LIN {X 0,Y 538.13,Z 595.444,A -85,B 0,C 180,E1 -4149.775,E2 -4149.775} C_VEL
LIN {X 0,Y 538.366,Z 585.113,A -85,B 0,C 180,E1 -4150.721,E2 -4150.721} C_VEL
LIN {X 0,Y 538.641,Z 573.919,A -85,B 0,C 180,E1 -4151.54,E2 -4151.54} C_VEL
LIN {X 0,Y 538.832,Z 561.69,A -85,B 0,C 180,E1 -4152.237,E2 -4152.237} C_VEL
LIN {X 0,Y 539.079,Z 549.655,A -85,B 0,C 180,E1 -4152.757,E2 -4152.757} C_VEL
LIN {X 0,Y 539.25,Z 536.276,A -85,B 0,C 180,E1 -4153.16,E2 -4153.16} C_VEL
LIN {X 0,Y 539.341,Z 523.449,A -85,B 0,C 180,E1 -4153.397,E2 -4153.397} C_VEL
LIN {X 0,Y 539.592,Z 428.794,A -85,B 0,C 180,E1 -4154.665,E2 -4154.665} C_VEL
LIN {X 0,Y 538.556,Z 421.341,A -85,B 0,C 180,E1 -4154.818,E2 -4154.818} C_VEL
LIN {X 0,Y 538.888,Z 398.914,A -85,B 0,C 180,E1 -4157.681,E2 -4157.681} C_VEL
LIN {X 0,Y 539.305,Z 376.337,A -85,B 0,C 180,E1 -4160.601,E2 -4160.601} C_VEL
LIN {X 0,Y 539.597,Z 359.195,A -85,B 0,C 180,E1 -4162.827,E2 -4162.827} C_VEL
LIN {X 0,Y 539.121,Z 355.573,A -85,B 0,C 180,E1 -4163.32,E2 -4163.32} C_VEL
LIN {X 0,Y 536.659,Z 349.989,A -85,B 0,C 180,E1 -4164.149,E2 -4164.149} C_VEL
LIN {X 0,Y 533.324,Z 343.375,A -85,B 0,C 180,E1 -4165.16,E2 -4165.16} C_VEL
LIN {X 0,Y 532.661,Z 341.028,A -85,B 0,C 180,E1 -4165.499,E2 -4165.499} C_VEL
LIN {X 0,Y 531.046,Z 333.084,A -85,B 0,C 180,E1 -4166.66,E2 -4166.66} C_VEL
LIN {X 0,Y 530.987,Z 332.967,A -85,B 0,C 180,E1 -4169.322,E2 -4169.322} C_VEL
LIN {X 0,Y 530.971,Z 332.971,A -85,B 0,C 180,E1 -4172.1,E2 -4172.1} C_VEL
LIN {X 0,Y 530.975,Z 332.968,A -85,B 0,C 180,E1 -4174.851,E2 -4174.851} C_VEL
LIN {X 0,Y 530.97,Z 332.966,A -85,B 0,C 180,E1 -4177.507,E2 -4177.507} C_VEL
LIN {X 0,Y 530.986,Z 332.97,A -85,B 0,C 180,E1 -4180.433,E2 -4180.433} C_VEL
LIN {X 0,Y 530.966,Z 332.964,A -85,B 0,C 180,E1 -4183.281,E2 -4183.281} C_VEL
LIN {X 0,Y 530.986,Z 332.959,A -85,B 0,C 180,E1 -4185.621,E2 -4185.621} C_VEL
LIN {X 0,Y 530.998,Z 332.964,A -85,B 0,C 180,E1 -4188.564,E2 -4188.564} C_VEL
LIN {X 0,Y 530.962,Z 332.967,A -85,B 0,C 180,E1 -4191.529,E2 -4191.529} C_VEL
LIN {X 0,Y 530.982,Z 332.968,A -85,B 0,C 180,E1 -4194.381,E2 -4194.381} C_VEL
LIN {X 0,Y 530.972,Z 332.964,A -85,B 0,C 180,E1 -4197.133,E2 -4197.133} C_VEL
LIN {X 0,Y 530.975,Z 332.967,A -85,B 0,C 180,E1 -4199.803,E2 -4199.803} C_VEL
LIN {X 0,Y 531.021,Z 332.964,A -85,B 0,C 180,E1 -4202.466,E2 -4202.466} C_VEL
LIN {X 0,Y 531.02,Z 332.968,A -85,B 0,C 180,E1 -4205.569,E2 -4205.569} C_VEL
LIN {X 0,Y 531.055,Z 333.297,A -85,B 0,C 180,E1 -4205.844,E2 -4205.844} C_VEL
LIN {X 0,Y 532.646,Z 342.082,A -85,B 0,C 180,E1 -4207.318,E2 -4207.318} C_VEL
LIN {X 0,Y 532.073,Z 361.559,A -85,B 0,C 180,E1 -4210.316,E2 -4210.316} C_VEL
LIN {X 0,Y 531.85,Z 372.04,A -85,B 0,C 180,E1 -4211.889,E2 -4211.889} C_VEL
LIN {X 0,Y 532.504,Z 375.809,A -85,B 0,C 180,E1 -4212.004,E2 -4212.004} C_VEL
LIN {X 0,Y 533.949,Z 384.074,A -85,B 0,C 180,E1 -4212.169,E2 -4212.169} C_VEL
LIN {X 0,Y 533.298,Z 508.609,A -85,B 0,C 180,E1 -4213.884,E2 -4213.884} C_VEL
LIN {X 0,Y 533.064,Z 523.105,A -85,B 0,C 180,E1 -4214.225,E2 -4214.225} C_VEL
LIN {X 0,Y 532.771,Z 537.785,A -85,B 0,C 180,E1 -4214.751,E2 -4214.751} C_VEL
LIN {X 0,Y 532.511,Z 550.755,A -85,B 0,C 180,E1 -4215.379,E2 -4215.379} C_VEL
LIN {X 0,Y 532.156,Z 561.953,A -85,B 0,C 180,E1 -4216.052,E2 -4216.052} C_VEL
LIN {X 0,Y 531.811,Z 573.767,A -85,B 0,C 180,E1 -4216.919,E2 -4216.919} C_VEL
LIN {X 0,Y 531.434,Z 586.265,A -85,B 0,C 180,E1 -4218.057,E2 -4218.057} C_VEL
LIN {X 0,Y 531.191,Z 595.879,A -85,B 0,C 180,E1 -4219.132,E2 -4219.132} C_VEL
LIN {X 0,Y 530.938,Z 603.182,A -85,B 0,C 180,E1 -4220.09,E2 -4220.09} C_VEL
LIN {X 0,Y 530.824,Z 609.461,A -85,B 0,C 180,E1 -4221.049,E2 -4221.049} C_VEL
LIN {X 0,Y 530.706,Z 614.868,A -85,B 0,C 180,E1 -4222.006,E2 -4222.006} C_VEL
LIN {X 0,Y 530.575,Z 620.295,A -85,B 0,C 180,E1 -4223.152,E2 -4223.152} C_VEL
LIN {X 0,Y 530.567,Z 624.738,A -85,B 0,C 180,E1 -4224.298,E2 -4224.298} C_VEL
LIN {X 0,Y 530.449,Z 628.286,A -85,B 0,C 180,E1 -4225.44,E2 -4225.44} C_VEL
LIN {X 0,Y 530.497,Z 630.208,A -85,B 0,C 180,E1 -4226.201,E2 -4226.201} C_VEL
LIN {X 0,Y 530.41,Z 632.929,A -85,B 0,C 180,E1 -4227.721,E2 -4227.721} C_VEL
LIN {X 0,Y 530.34,Z 634.237,A -85,B 0,C 180,E1 -4229.24,E2 -4229.24} C_VEL
LIN {X 0,Y 530.342,Z 634.496,A -85,B 0,C 180,E1 -4229.999,E2 -4229.999} C_VEL
LIN {X 0,Y 530.357,Z 633.834,A -85,B 0,C 180,E1 -4231.518,E2 -4231.518} C_VEL
LIN {X 0,Y 530.451,Z 631.843,A -85,B 0,C 180,E1 -4233.037,E2 -4233.037} C_VEL
LIN {X 0,Y 530.497,Z 630.435,A -85,B 0,C 180,E1 -4233.797,E2 -4233.797} C_VEL
LIN {X 0,Y 530.514,Z 626.296,A -85,B 0,C 180,E1 -4235.32,E2 -4235.32} C_VEL
LIN {X 0,Y 530.555,Z 623.773,A -85,B 0,C 180,E1 -4236.082,E2 -4236.082} C_VEL
LIN {X 0,Y 530.584,Z 619.088,A -85,B 0,C 180,E1 -4237.228,E2 -4237.228} C_VEL
LIN {X 0,Y 530.774,Z 612.262,A -85,B 0,C 180,E1 -4238.566,E2 -4238.566} C_VEL
LIN {X 0,Y 530.895,Z 605.147,A -85,B 0,C 180,E1 -4239.716,E2 -4239.716} C_VEL
LIN {X 0,Y 531.097,Z 598.173,A -85,B 0,C 180,E1 -4240.675,E2 -4240.675} C_VEL
LIN {X 0,Y 531.373,Z 589.079,A -85,B 0,C 180,E1 -4241.733,E2 -4241.733} C_VEL
LIN {X 0,Y 531.625,Z 580.332,A -85,B 0,C 180,E1 -4242.598,E2 -4242.598} C_VEL
LIN {X 0,Y 531.914,Z 569.995,A -85,B 0,C 180,E1 -4243.465,E2 -4243.465} C_VEL
LIN {X 0,Y 532.249,Z 558.953,A -85,B 0,C 180,E1 -4244.236,E2 -4244.236} C_VEL
LIN {X 0,Y 532.596,Z 544.118,A -85,B 0,C 180,E1 -4245.057,E2 -4245.057} C_VEL
LIN {X 0,Y 532.936,Z 531.187,A -85,B 0,C 180,E1 -4245.595,E2 -4245.595} C_VEL
LIN {X 0,Y 533.153,Z 518.305,A -85,B 0,C 180,E1 -4245.992,E2 -4245.992} C_VEL
LIN {X 0,Y 533.333,Z 505.438,A -85,B 0,C 180,E1 -4246.26,E2 -4246.26} C_VEL
LIN {X 0,Y 533.841,Z 382.931,A -85,B 0,C 180,E1 -4247.941,E2 -4247.941} C_VEL
LIN {X 0,Y 531.872,Z 372.407,A -85,B 0,C 180,E1 -4248.173,E2 -4248.173} C_VEL
LIN {X 0,Y 531.921,Z 368.698,A -85,B 0,C 180,E1 -4248.686,E2 -4248.686} C_VEL
LIN {X 0,Y 532.441,Z 349.078,A -85,B 0,C 180,E1 -4251.689,E2 -4251.689} C_VEL
LIN {X 0,Y 532.622,Z 341.232,A -85,B 0,C 180,E1 -4252.906,E2 -4252.906} C_VEL
LIN {X 0,Y 531.016,Z 333.185,A -85,B 0,C 180,E1 -4254.273,E2 -4254.273} C_VEL
LIN {X 0,Y 531.014,Z 332.957,A -85,B 0,C 180,E1 -4255.896,E2 -4255.896} C_VEL
LIN {X 0,Y 530.998,Z 332.957,A -85,B 0,C 180,E1 -4258.454,E2 -4258.454} C_VEL
LIN {X 0,Y 530.965,Z 332.967,A -85,B 0,C 180,E1 -4261.077,E2 -4261.077} C_VEL
LIN {X 0,Y 530.99,Z 332.966,A -85,B 0,C 180,E1 -4263.771,E2 -4263.771} C_VEL
LIN {X 0,Y 530.965,Z 332.968,A -85,B 0,C 180,E1 -4266.556,E2 -4266.556} C_VEL
LIN {X 0,Y 531.002,Z 332.964,A -85,B 0,C 180,E1 -4269.856,E2 -4269.856} C_VEL
LIN {X 0,Y 530.977,Z 332.967,A -85,B 0,C 180,E1 -4272.455,E2 -4272.455} C_VEL
LIN {X 0,Y 530.982,Z 332.962,A -85,B 0,C 180,E1 -4275.62,E2 -4275.62} C_VEL
LIN {X 0,Y 531.013,Z 332.961,A -85,B 0,C 180,E1 -4278.566,E2 -4278.566} C_VEL
LIN {X 0,Y 530.953,Z 332.967,A -85,B 0,C 180,E1 -4281.529,E2 -4281.529} C_VEL
LIN {X 0,Y 530.974,Z 332.964,A -85,B 0,C 180,E1 -4284.381,E2 -4284.381} C_VEL
LIN {X 0,Y 530.967,Z 332.968,A -85,B 0,C 180,E1 -4287.133,E2 -4287.133} C_VEL
LIN {X 0,Y 530.977,Z 332.958,A -85,B 0,C 180,E1 -4289.803,E2 -4289.803} C_VEL
LIN {X 0,Y 531.009,Z 332.953,A -85,B 0,C 180,E1 -4292.465,E2 -4292.465} C_VEL
LIN {X 0,Y 531.001,Z 332.962,A -85,B 0,C 180,E1 -4294.942,E2 -4294.942} C_VEL
LIN {X 0,Y 530.982,Z 332.963,A -85,B 0,C 180,E1 -4297.893,E2 -4297.893} C_VEL
LIN {X 0,Y 530.988,Z 332.963,A -85,B 0,C 180,E1 -4300.677,E2 -4300.677} C_VEL
LIN {X 0,Y 530.985,Z 332.968,A -85,B 0,C 180,E1 -4303.071,E2 -4303.071} C_VEL
LIN {X 0,Y 531.03,Z 332.963,A -85,B 0,C 180,E1 -4305.436,E2 -4305.436} C_VEL
LIN {X 0,Y 531.043,Z 332.956,A -85,B 0,C 180,E1 -4308.55,E2 -4308.55} C_VEL
LIN {X 0,Y 531.052,Z 332.956,A -85,B 0,C 180,E1 -4311.629,E2 -4311.629} C_VEL
LIN {X 0,Y 531.132,Z 332.947,A -85,B 0,C 180,E1 -4314.685,E2 -4314.685} C_VEL
LIN {X 0,Y 531.131,Z 332.944,A -85,B 0,C 180,E1 -4317.725,E2 -4317.725} C_VEL
LIN {X 0,Y 531.149,Z 332.948,A -85,B 0,C 180,E1 -4320.758,E2 -4320.758} C_VEL
LIN {X 0,Y 531.103,Z 332.952,A -85,B 0,C 180,E1 -4323.034,E2 -4323.034} C_VEL
LIN {X 0,Y 531.076,Z 332.952,A -85,B 0,C 180,E1 -4326.077,E2 -4326.077} C_VEL
LIN {X 0,Y 531.028,Z 332.957,A -85,B 0,C 180,E1 -4329.138,E2 -4329.138} C_VEL
LIN {X 0,Y 531.051,Z 332.954,A -85,B 0,C 180,E1 -4331.678,E2 -4331.678} C_VEL
LIN {X 0,Y 531.019,Z 332.959,A -85,B 0,C 180,E1 -4334.956,E2 -4334.956} C_VEL
LIN {X 0,Y 531.006,Z 332.96,A -85,B 0,C 180,E1 -4337.723,E2 -4337.723} C_VEL
LIN {X 0,Y 530.995,Z 332.963,A -85,B 0,C 180,E1 -4340.938,E2 -4340.938} C_VEL
LIN {X 0,Y 530.998,Z 332.964,A -85,B 0,C 180,E1 -4344.046,E2 -4344.046} C_VEL
LIN {X 0,Y 531.002,Z 332.959,A -85,B 0,C 180,E1 -4346.744,E2 -4346.744} C_VEL
LIN {X 0,Y 530.973,Z 332.952,A -85,B 0,C 180,E1 -4349.323,E2 -4349.323} C_VEL
LIN {X 0,Y 530.972,Z 332.966,A -85,B 0,C 180,E1 -4352.104,E2 -4352.104} C_VEL
LIN {X 0,Y 530.982,Z 332.965,A -85,B 0,C 180,E1 -4354.855,E2 -4354.855} C_VEL
LIN {X 0,Y 530.958,Z 332.958,A -85,B 0,C 180,E1 -4357.508,E2 -4357.508} C_VEL
LIN {X 0,Y 531.02,Z 332.966,A -85,B 0,C 180,E1 -4360.429,E2 -4360.429} C_VEL
LIN {X 0,Y 530.961,Z 332.965,A -85,B 0,C 180,E1 -4363.495,E2 -4363.495} C_VEL
LIN {X 0,Y 530.959,Z 332.971,A -85,B 0,C 180,E1 -4366.507,E2 -4366.507} C_VEL
LIN {X 0,Y 531.021,Z 332.96,A -85,B 0,C 180,E1 -4369.572,E2 -4369.572} C_VEL
LIN {X 0,Y 530.964,Z 332.968,A -85,B 0,C 180,E1 -4372.578,E2 -4372.578} C_VEL
LIN {X 0,Y 531.001,Z 332.963,A -85,B 0,C 180,E1 -4375.313,E2 -4375.313} C_VEL
LIN {X 0,Y 530.98,Z 332.972,A -85,B 0,C 180,E1 -4378.034,E2 -4378.034} C_VEL
LIN {X 0,Y 531.004,Z 332.951,A -85,B 0,C 180,E1 -4380.872,E2 -4380.872} C_VEL
LIN {X 0,Y 531.01,Z 332.966,A -85,B 0,C 180,E1 -4383.258,E2 -4383.258} C_VEL
LIN {X 0,Y 531.009,Z 333.054,A -85,B 0,C 180,E1 -4385.726,E2 -4385.726} C_VEL
LIN {X 0,Y 532.599,Z 340.946,A -85,B 0,C 180,E1 -4387.092,E2 -4387.092} C_VEL
LIN {X 0,Y 532.226,Z 357.451,A -85,B 0,C 180,E1 -4389.644,E2 -4389.644} C_VEL
LIN {X 0,Y 531.845,Z 372.091,A -85,B 0,C 180,E1 -4391.849,E2 -4391.849} C_VEL
LIN {X 0,Y 532.716,Z 376.892,A -85,B 0,C 180,E1 -4391.982,E2 -4391.982} C_VEL
LIN {X 0,Y 533.891,Z 384.047,A -85,B 0,C 180,E1 -4392.122,E2 -4392.122} C_VEL
LIN {X 0,Y 533.278,Z 508.696,A -85,B 0,C 180,E1 -4393.836,E2 -4393.836} C_VEL
LIN {X 0,Y 533.082,Z 523.313,A -85,B 0,C 180,E1 -4394.188,E2 -4394.188} C_VEL
LIN {X 0,Y 532.852,Z 536.169,A -85,B 0,C 180,E1 -4394.639,E2 -4394.639} C_VEL
LIN {X 0,Y 532.521,Z 549.89,A -85,B 0,C 180,E1 -4395.284,E2 -4395.284} C_VEL
LIN {X 0,Y 532.144,Z 562.69,A -85,B 0,C 180,E1 -4396.054,E2 -4396.054} C_VEL
LIN {X 0,Y 531.803,Z 574.318,A -85,B 0,C 180,E1 -4396.921,E2 -4396.921} C_VEL
LIN {X 0,Y 531.453,Z 585.317,A -85,B 0,C 180,E1 -4397.917,E2 -4397.917} C_VEL
LIN {X 0,Y 531.234,Z 594.715,A -85,B 0,C 180,E1 -4398.942,E2 -4398.942} C_VEL
LIN {X 0,Y 530.935,Z 603.563,A -85,B 0,C 180,E1 -4400.092,E2 -4400.092} C_VEL
LIN {X 0,Y 530.774,Z 612.04,A -85,B 0,C 180,E1 -4401.434,E2 -4401.434} C_VEL
LIN {X 0,Y 530.585,Z 618.866,A -85,B 0,C 180,E1 -4402.772,E2 -4402.772} C_VEL
LIN {X 0,Y 530.584,Z 624.962,A -85,B 0,C 180,E1 -4404.3,E2 -4404.3} C_VEL
LIN {X 0,Y 530.449,Z 628.449,A -85,B 0,C 180,E1 -4405.441,E2 -4405.441} C_VEL
LIN {X 0,Y 530.452,Z 631.838,A -85,B 0,C 180,E1 -4406.963,E2 -4406.963} C_VEL
LIN {X 0,Y 530.357,Z 633.838,A -85,B 0,C 180,E1 -4408.482,E2 -4408.482} C_VEL
LIN {X 0,Y 530.341,Z 634.5,A -85,B 0,C 180,E1 -4410.001,E2 -4410.001} C_VEL
LIN {X 0,Y 530.357,Z 633.834,A -85,B 0,C 180,E1 -4411.52,E2 -4411.52} C_VEL
LIN {X 0,Y 530.452,Z 631.83,A -85,B 0,C 180,E1 -4413.039,E2 -4413.039} C_VEL
LIN {X 0,Y 530.449,Z 628.441,A -85,B 0,C 180,E1 -4414.56,E2 -4414.56} C_VEL
LIN {X 0,Y 530.561,Z 623.565,A -85,B 0,C 180,E1 -4416.084,E2 -4416.084} C_VEL
LIN {X 0,Y 530.642,Z 617.05,A -85,B 0,C 180,E1 -4417.612,E2 -4417.612} C_VEL
LIN {X 0,Y 530.812,Z 609.797,A -85,B 0,C 180,E1 -4418.951,E2 -4418.951} C_VEL
LIN {X 0,Y 531.018,Z 600.815,A -85,B 0,C 180,E1 -4420.293,E2 -4420.293} C_VEL
LIN {X 0,Y 531.312,Z 591.383,A -85,B 0,C 180,E1 -4421.445,E2 -4421.445} C_VEL
LIN {X 0,Y 531.586,Z 580.942,A -85,B 0,C 180,E1 -4422.504,E2 -4422.504} C_VEL
LIN {X 0,Y 531.951,Z 569.413,A -85,B 0,C 180,E1 -4423.466,E2 -4423.466} C_VEL
LIN {X 0,Y 532.284,Z 558.201,A -85,B 0,C 180,E1 -4424.237,E2 -4424.237} C_VEL
LIN {X 0,Y 532.613,Z 546.119,A -85,B 0,C 180,E1 -4424.911,E2 -4424.911} C_VEL
LIN {X 0,Y 532.939,Z 533.26,A -85,B 0,C 180,E1 -4425.473,E2 -4425.473} C_VEL
LIN {X 0,Y 533.092,Z 519.619,A -85,B 0,C 180,E1 -4425.916,E2 -4425.916} C_VEL
LIN {X 0,Y 533.304,Z 505.572,A -85,B 0,C 180,E1 -4426.214,E2 -4426.214} C_VEL
LIN {X 0,Y 533.922,Z 383.42,A -85,B 0,C 180,E1 -4427.886,E2 -4427.886} C_VEL
LIN {X 0,Y 531.879,Z 372.396,A -85,B 0,C 180,E1 -4428.129,E2 -4428.129} C_VEL
LIN {X 0,Y 531.938,Z 367.082,A -85,B 0,C 180,E1 -4428.887,E2 -4428.887} C_VEL
LIN {X 0,Y 532.429,Z 348.776,A -85,B 0,C 180,E1 -4431.692,E2 -4431.692} C_VEL
LIN {X 0,Y 532.605,Z 340.932,A -85,B 0,C 180,E1 -4432.909,E2 -4432.909} C_VEL
LIN {X 0,Y 531.04,Z 333.202,A -85,B 0,C 180,E1 -4434.222,E2 -4434.222} C_VEL
LIN {X 0,Y 531.011,Z 332.961,A -85,B 0,C 180,E1 -4435.058,E2 -4435.058} C_VEL
LIN {X 0,Y 531.022,Z 332.964,A -85,B 0,C 180,E1 -4437.596,E2 -4437.596} C_VEL
LIN {X 0,Y 530.979,Z 332.968,A -85,B 0,C 180,E1 -4440.646,E2 -4440.646} C_VEL
LIN {X 0,Y 530.995,Z 332.968,A -85,B 0,C 180,E1 -4443.773,E2 -4443.773} C_VEL
LIN {X 0,Y 530.974,Z 332.968,A -85,B 0,C 180,E1 -4446.558,E2 -4446.558} C_VEL
LIN {X 0,Y 530.983,Z 332.971,A -85,B 0,C 180,E1 -4449.854,E2 -4449.854} C_VEL
LIN {X 0,Y 530.982,Z 332.966,A -85,B 0,C 180,E1 -4452.457,E2 -4452.457} C_VEL
LIN {X 0,Y 530.987,Z 332.969,A -85,B 0,C 180,E1 -4455.622,E2 -4455.622} C_VEL
LIN {X 0,Y 531.001,Z 332.964,A -85,B 0,C 180,E1 -4458.565,E2 -4458.565} C_VEL
LIN {X 0,Y 530.961,Z 332.973,A -85,B 0,C 180,E1 -4461.53,E2 -4461.53} C_VEL
LIN {X 0,Y 530.958,Z 332.969,A -85,B 0,C 180,E1 -4464.38,E2 -4464.38} C_VEL
LIN {X 0,Y 530.972,Z 332.97,A -85,B 0,C 180,E1 -4467.134,E2 -4467.134} C_VEL
LIN {X 0,Y 530.974,Z 332.973,A -85,B 0,C 180,E1 -4469.803,E2 -4469.803} C_VEL
LIN {X 0,Y 531.02,Z 332.964,A -85,B 0,C 180,E1 -4472.467,E2 -4472.467} C_VEL
LIN {X 0,Y 531.038,Z 333.152,A -85,B 0,C 180,E1 -4473.857,E2 -4473.857} C_VEL
LIN {X 0,Y 532.577,Z 341.879,A -85,B 0,C 180,E1 -4475.021,E2 -4475.021} C_VEL
LIN {X 0,Y 532.429,Z 361.787,A -85,B 0,C 180,E1 -4477.518,E2 -4477.518} C_VEL
LIN {X 0,Y 532.201,Z 380.833,A -85,B 0,C 180,E1 -4479.919,E2 -4479.919} C_VEL
LIN {X 0,Y 531.914,Z 397.433,A -85,B 0,C 180,E1 -4482.049,E2 -4482.049} C_VEL
LIN {X 0,Y 531.596,Z 417.775,A -85,B 0,C 180,E1 -4484.668,E2 -4484.668} C_VEL
LIN {X 0,Y 531.551,Z 421.298,A -85,B 0,C 180,E1 -4485.083,E2 -4485.083} C_VEL
LIN {X 0,Y 532.8,Z 431.144,A -85,B 0,C 180,E1 -4485.276,E2 -4485.276} C_VEL
LIN {X 0,Y 532.344,Z 530.888,A -85,B 0,C 180,E1 -4486.666,E2 -4486.666} C_VEL
LIN {X 0,Y 532.209,Z 543.359,A -85,B 0,C 180,E1 -4486.979,E2 -4486.979} C_VEL
LIN {X 0,Y 531.963,Z 556.15,A -85,B 0,C 180,E1 -4487.458,E2 -4487.458} C_VEL
LIN {X 0,Y 531.746,Z 568.289,A -85,B 0,C 180,E1 -4488.076,E2 -4488.076} C_VEL
LIN {X 0,Y 531.523,Z 578.707,A -85,B 0,C 180,E1 -4488.754,E2 -4488.754} C_VEL
LIN {X 0,Y 531.25,Z 589.326,A -85,B 0,C 180,E1 -4489.616,E2 -4489.616} C_VEL
LIN {X 0,Y 531.006,Z 599.735,A -85,B 0,C 180,E1 -4490.669,E2 -4490.669} C_VEL
LIN {X 0,Y 530.857,Z 607.422,A -85,B 0,C 180,E1 -4491.626,E2 -4491.626} C_VEL
LIN {X 0,Y 530.673,Z 614.918,A -85,B 0,C 180,E1 -4492.772,E2 -4492.772} C_VEL
LIN {X 0,Y 530.611,Z 620.932,A -85,B 0,C 180,E1 -4493.918,E2 -4493.918} C_VEL
LIN {X 0,Y 530.459,Z 625.687,A -85,B 0,C 180,E1 -4495.06,E2 -4495.06} C_VEL
LIN {X 0,Y 530.517,Z 629.324,A -85,B 0,C 180,E1 -4496.202,E2 -4496.202} C_VEL
LIN {X 0,Y 530.458,Z 631.196,A -85,B 0,C 180,E1 -4496.962,E2 -4496.962} C_VEL
LIN {X 0,Y 530.411,Z 632.631,A -85,B 0,C 180,E1 -4497.722,E2 -4497.722} C_VEL
LIN {X 0,Y 530.344,Z 634.256,A -85,B 0,C 180,E1 -4499.241,E2 -4499.241} C_VEL
LIN {X 0,Y 530.343,Z 634.497,A -85,B 0,C 180,E1 -4500,E2 -4500} C_VEL
LIN {X 0,Y 530.344,Z 634.312,A -85,B 0,C 180,E1 -4500.759,E2 -4500.759} C_VEL
LIN {X 0,Y 530.41,Z 632.763,A -85,B 0,C 180,E1 -4502.278,E2 -4502.278} C_VEL
LIN {X 0,Y 530.458,Z 631.4,A -85,B 0,C 180,E1 -4503.038,E2 -4503.038} C_VEL
LIN {X 0,Y 530.523,Z 628.526,A -85,B 0,C 180,E1 -4504.178,E2 -4504.178} C_VEL
LIN {X 0,Y 530.524,Z 624.616,A -85,B 0,C 180,E1 -4505.321,E2 -4505.321} C_VEL
LIN {X 0,Y 530.606,Z 618.542,A -85,B 0,C 180,E1 -4506.66,E2 -4506.66} C_VEL
LIN {X 0,Y 530.759,Z 611.965,A -85,B 0,C 180,E1 -4507.801,E2 -4507.801} C_VEL
LIN {X 0,Y 530.907,Z 603.733,A -85,B 0,C 180,E1 -4508.948,E2 -4508.948} C_VEL
LIN {X 0,Y 531.098,Z 595.256,A -85,B 0,C 180,E1 -4509.906,E2 -4509.906} C_VEL
LIN {X 0,Y 531.377,Z 584.867,A -85,B 0,C 180,E1 -4510.864,E2 -4510.864} C_VEL
LIN {X 0,Y 531.636,Z 574.017,A -85,B 0,C 180,E1 -4511.667,E2 -4511.667} C_VEL
LIN {X 0,Y 531.832,Z 563.162,A -85,B 0,C 180,E1 -4512.303,E2 -4512.303} C_VEL
LIN {X 0,Y 532.104,Z 550.353,A -85,B 0,C 180,E1 -4512.879,E2 -4512.879} C_VEL
LIN {X 0,Y 532.292,Z 537.451,A -85,B 0,C 180,E1 -4513.287,E2 -4513.287} C_VEL
LIN {X 0,Y 532.416,Z 523.828,A -85,B 0,C 180,E1 -4513.551,E2 -4513.551} C_VEL
LIN {X 0,Y 532.692,Z 429.041,A -85,B 0,C 180,E1 -4514.851,E2 -4514.851} C_VEL
LIN {X 0,Y 531.559,Z 421.111,A -85,B 0,C 180,E1 -4515.025,E2 -4515.025} C_VEL
LIN {X 0,Y 532.009,Z 396.96,A -85,B 0,C 180,E1 -4518.151,E2 -4518.151} C_VEL
LIN {X 0,Y 532.469,Z 371.438,A -85,B 0,C 180,E1 -4521.486,E2 -4521.486} C_VEL
LIN {X 0,Y 532.901,Z 351.257,A -85,B 0,C 180,E1 -4524.132,E2 -4524.132} C_VEL
LIN {X 0,Y 532.82,Z 341.844,A -85,B 0,C 180,E1 -4525.384,E2 -4525.384} C_VEL
LIN {X 0,Y 532.661,Z 341.028,A -85,B 0,C 180,E1 -4525.499,E2 -4525.499} C_VEL
LIN {X 0,Y 531.517,Z 338.82,A -85,B 0,C 180,E1 -4525.844,E2 -4525.844} C_VEL
LIN {X 0,Y 528.005,Z 335.837,A -85,B 0,C 180,E1 -4526.408,E2 -4526.408} C_VEL
LIN {X 0,Y 524.989,Z 334.278,A -85,B 0,C 180,E1 -4526.961,E2 -4526.961} C_VEL
LIN {X 0,Y 523.994,Z 333.853,A -85,B 0,C 180,E1 -4527.38,E2 -4527.38} C_VEL
LIN {X 0,Y 523.97,Z 333.843,A -85,B 0,C 180,E1 -4527.453,E2 -4527.453} C_VEL
LIN {X 0,Y 523.961,Z 333.846,A -85,B 0,C 180,E1 -4530.644,E2 -4530.644} C_VEL
LIN {X 0,Y 523.964,Z 333.84,A -85,B 0,C 180,E1 -4533.734,E2 -4533.734} C_VEL
LIN {X 0,Y 523.909,Z 333.854,A -85,B 0,C 180,E1 -4536.401,E2 -4536.401} C_VEL
LIN {X 0,Y 523.925,Z 333.844,A -85,B 0,C 180,E1 -4539.085,E2 -4539.085} C_VEL
LIN {X 0,Y 523.956,Z 333.846,A -85,B 0,C 180,E1 -4542.119,E2 -4542.119} C_VEL
LIN {X 0,Y 523.95,Z 333.833,A -85,B 0,C 180,E1 -4545.31,E2 -4545.31} C_VEL
LIN {X 0,Y 523.961,Z 333.839,A -85,B 0,C 180,E1 -4548.689,E2 -4548.689} C_VEL
LIN {X 0,Y 523.922,Z 333.842,A -85,B 0,C 180,E1 -4551.08,E2 -4551.08} C_VEL
LIN {X 0,Y 523.929,Z 333.847,A -85,B 0,C 180,E1 -4553.827,E2 -4553.827} C_VEL
LIN {X 0,Y 523.947,Z 333.84,A -85,B 0,C 180,E1 -4556.635,E2 -4556.635} C_VEL
LIN {X 0,Y 523.961,Z 333.842,A -85,B 0,C 180,E1 -4559.355,E2 -4559.355} C_VEL
LIN {X 0,Y 523.984,Z 333.843,A -85,B 0,C 180,E1 -4562.281,E2 -4562.281} C_VEL
LIN {X 0,Y 523.999,Z 333.841,A -85,B 0,C 180,E1 -4565.431,E2 -4565.431} C_VEL
LIN {X 0,Y 524.02,Z 334.225,A -85,B 0,C 180,E1 -4565.652,E2 -4565.652} C_VEL
LIN {X 0,Y 525.728,Z 343.262,A -85,B 0,C 180,E1 -4567.189,E2 -4567.189} C_VEL
LIN {X 0,Y 525.185,Z 361.563,A -85,B 0,C 180,E1 -4570.047,E2 -4570.047} C_VEL
LIN {X 0,Y 524.95,Z 372.299,A -85,B 0,C 180,E1 -4571.664,E2 -4571.664} C_VEL
LIN {X 0,Y 527.182,Z 385.222,A -85,B 0,C 180,E1 -4571.948,E2 -4571.948} C_VEL
LIN {X 0,Y 526.486,Z 508.798,A -85,B 0,C 180,E1 -4573.67,E2 -4573.67} C_VEL
LIN {X 0,Y 526.238,Z 523.501,A -85,B 0,C 180,E1 -4574.027,E2 -4574.027} C_VEL
LIN {X 0,Y 525.937,Z 537.794,A -85,B 0,C 180,E1 -4574.548,E2 -4574.548} C_VEL
LIN {X 0,Y 525.639,Z 550.797,A -85,B 0,C 180,E1 -4575.184,E2 -4575.184} C_VEL
LIN {X 0,Y 525.197,Z 563.428,A -85,B 0,C 180,E1 -4575.962,E2 -4575.962} C_VEL
LIN {X 0,Y 524.769,Z 576.118,A -85,B 0,C 180,E1 -4576.937,E2 -4576.937} C_VEL
LIN {X 0,Y 524.439,Z 586.655,A -85,B 0,C 180,E1 -4577.934,E2 -4577.934} C_VEL
LIN {X 0,Y 524.177,Z 595.919,A -85,B 0,C 180,E1 -4578.984,E2 -4578.984} C_VEL
LIN {X 0,Y 523.892,Z 604.544,A -85,B 0,C 180,E1 -4580.151,E2 -4580.151} C_VEL
LIN {X 0,Y 523.715,Z 611.747,A -85,B 0,C 180,E1 -4581.316,E2 -4581.316} C_VEL
LIN {X 0,Y 523.51,Z 618.659,A -85,B 0,C 180,E1 -4582.672,E2 -4582.672} C_VEL
LIN {X 0,Y 523.481,Z 624.758,A -85,B 0,C 180,E1 -4584.22,E2 -4584.22} C_VEL
LIN {X 0,Y 523.353,Z 628.307,A -85,B 0,C 180,E1 -4585.378,E2 -4585.378} C_VEL
LIN {X 0,Y 523.42,Z 630.219,A -85,B 0,C 180,E1 -4586.15,E2 -4586.15} C_VEL
LIN {X 0,Y 523.334,Z 632.938,A -85,B 0,C 180,E1 -4587.69,E2 -4587.69} C_VEL
LIN {X 0,Y 523.246,Z 634.249,A -85,B 0,C 180,E1 -4589.229,E2 -4589.229} C_VEL
LIN {X 0,Y 523.245,Z 634.496,A -85,B 0,C 180,E1 -4589.999,E2 -4589.999} C_VEL
LIN {X 0,Y 523.271,Z 633.842,A -85,B 0,C 180,E1 -4591.538,E2 -4591.538} C_VEL
LIN {X 0,Y 523.362,Z 631.856,A -85,B 0,C 180,E1 -4593.078,E2 -4593.078} C_VEL
LIN {X 0,Y 523.419,Z 630.432,A -85,B 0,C 180,E1 -4593.848,E2 -4593.848} C_VEL
LIN {X 0,Y 523.448,Z 626.311,A -85,B 0,C 180,E1 -4595.392,E2 -4595.392} C_VEL
LIN {X 0,Y 523.487,Z 622.28,A -85,B 0,C 180,E1 -4596.546,E2 -4596.546} C_VEL
LIN {X 0,Y 523.567,Z 617.247,A -85,B 0,C 180,E1 -4597.713,E2 -4597.713} C_VEL
LIN {X 0,Y 523.728,Z 611.153,A -85,B 0,C 180,E1 -4598.876,E2 -4598.876} C_VEL
LIN {X 0,Y 523.879,Z 603.841,A -85,B 0,C 180,E1 -4600.043,E2 -4600.043} C_VEL
LIN {X 0,Y 524.227,Z 595.095,A -85,B 0,C 180,E1 -4601.208,E2 -4601.208} C_VEL
LIN {X 0,Y 524.524,Z 584.461,A -85,B 0,C 180,E1 -4602.378,E2 -4602.378} C_VEL
LIN {X 0,Y 524.888,Z 572.502,A -85,B 0,C 180,E1 -4603.452,E2 -4603.452} C_VEL
LIN {X 0,Y 525.295,Z 560.448,A -85,B 0,C 180,E1 -4604.329,E2 -4604.329} C_VEL
LIN {X 0,Y 525.689,Z 547.07,A -85,B 0,C 180,E1 -4605.11,E2 -4605.11} C_VEL
LIN {X 0,Y 526.078,Z 533.368,A -85,B 0,C 180,E1 -4605.72,E2 -4605.72} C_VEL
LIN {X 0,Y 526.304,Z 520.05,A -85,B 0,C 180,E1 -4606.159,E2 -4606.159} C_VEL
LIN {X 0,Y 526.524,Z 505.4,A -85,B 0,C 180,E1 -4606.477,E2 -4606.477} C_VEL
LIN {X 0,Y 527.096,Z 383.792,A -85,B 0,C 180,E1 -4608.165,E2 -4608.165} C_VEL
LIN {X 0,Y 524.939,Z 372.25,A -85,B 0,C 180,E1 -4608.43,E2 -4608.43} C_VEL
LIN {X 0,Y 525.365,Z 354.306,A -85,B 0,C 180,E1 -4611.172,E2 -4611.172} C_VEL
LIN {X 0,Y 525.678,Z 342.534,A -85,B 0,C 180,E1 -4613.019,E2 -4613.019} C_VEL
LIN {X 0,Y 523.987,Z 333.966,A -85,B 0,C 180,E1 -4614.514,E2 -4614.514} C_VEL
LIN {X 0,Y 523.956,Z 333.843,A -85,B 0,C 180,E1 -4617.131,E2 -4617.131} C_VEL
LIN {X 0,Y 523.955,Z 333.832,A -85,B 0,C 180,E1 -4619.754,E2 -4619.754} C_VEL
LIN {X 0,Y 523.938,Z 333.844,A -85,B 0,C 180,E1 -4622.448,E2 -4622.448} C_VEL
LIN {X 0,Y 523.933,Z 333.842,A -85,B 0,C 180,E1 -4625.224,E2 -4625.224} C_VEL
LIN {X 0,Y 523.913,Z 333.851,A -85,B 0,C 180,E1 -4628.1,E2 -4628.1} C_VEL
LIN {X 0,Y 523.956,Z 333.837,A -85,B 0,C 180,E1 -4631.089,E2 -4631.089} C_VEL
LIN {X 0,Y 523.935,Z 333.839,A -85,B 0,C 180,E1 -4634.227,E2 -4634.227} C_VEL
LIN {X 0,Y 523.921,Z 333.841,A -85,B 0,C 180,E1 -4636.833,E2 -4636.833} C_VEL
LIN {X 0,Y 523.963,Z 333.839,A -85,B 0,C 180,E1 -4638.91,E2 -4638.91} C_VEL
LIN {X 0,Y 523.91,Z 333.839,A -85,B 0,C 180,E1 -4641.897,E2 -4641.897} C_VEL
LIN {X 0,Y 523.931,Z 333.841,A -85,B 0,C 180,E1 -4644.908,E2 -4644.908} C_VEL
LIN {X 0,Y 523.935,Z 333.847,A -85,B 0,C 180,E1 -4647.677,E2 -4647.677} C_VEL
LIN {X 0,Y 523.961,Z 333.824,A -85,B 0,C 180,E1 -4650.672,E2 -4650.672} C_VEL
LIN {X 0,Y 523.969,Z 333.842,A -85,B 0,C 180,E1 -4653.728,E2 -4653.728} C_VEL
LIN {X 0,Y 523.941,Z 333.841,A -85,B 0,C 180,E1 -4656.271,E2 -4656.271} C_VEL
LIN {X 0,Y 523.944,Z 333.838,A -85,B 0,C 180,E1 -4658.766,E2 -4658.766} C_VEL
LIN {X 0,Y 523.945,Z 333.846,A -85,B 0,C 180,E1 -4661.22,E2 -4661.22} C_VEL
LIN {X 0,Y 523.933,Z 333.841,A -85,B 0,C 180,E1 -4663.639,E2 -4663.639} C_VEL
LIN {X 0,Y 523.936,Z 333.84,A -85,B 0,C 180,E1 -4666.028,E2 -4666.028} C_VEL
LIN {X 0,Y 524.002,Z 333.838,A -85,B 0,C 180,E1 -4669.177,E2 -4669.177} C_VEL
LIN {X 0,Y 524.019,Z 333.829,A -85,B 0,C 180,E1 -4672.292,E2 -4672.292} C_VEL
LIN {X 0,Y 524.09,Z 333.824,A -85,B 0,C 180,E1 -4674.614,E2 -4674.614} C_VEL
LIN {X 0,Y 524.103,Z 333.82,A -85,B 0,C 180,E1 -4677.694,E2 -4677.694} C_VEL
LIN {X 0,Y 524.118,Z 333.824,A -85,B 0,C 180,E1 -4680.768,E2 -4680.768} C_VEL
LIN {X 0,Y 524.069,Z 333.827,A -85,B 0,C 180,E1 -4683.075,E2 -4683.075} C_VEL
LIN {X 0,Y 524.037,Z 333.829,A -85,B 0,C 180,E1 -4686.159,E2 -4686.159} C_VEL
LIN {X 0,Y 523.996,Z 333.831,A -85,B 0,C 180,E1 -4689.262,E2 -4689.262} C_VEL
LIN {X 0,Y 524.013,Z 333.83,A -85,B 0,C 180,E1 -4691.751,E2 -4691.751} C_VEL
LIN {X 0,Y 523.983,Z 333.834,A -85,B 0,C 180,E1 -4695.053,E2 -4695.053} C_VEL
LIN {X 0,Y 523.954,Z 333.839,A -85,B 0,C 180,E1 -4697.969,E2 -4697.969} C_VEL
LIN {X 0,Y 523.963,Z 333.842,A -85,B 0,C 180,E1 -4700.41,E2 -4700.41} C_VEL
LIN {X 0,Y 523.935,Z 333.846,A -85,B 0,C 180,E1 -4702.892,E2 -4702.892} C_VEL
LIN {X 0,Y 523.976,Z 333.837,A -85,B 0,C 180,E1 -4706.021,E2 -4706.021} C_VEL
LIN {X 0,Y 523.931,Z 333.831,A -85,B 0,C 180,E1 -4708.875,E2 -4708.875} C_VEL
LIN {X 0,Y 523.922,Z 333.84,A -85,B 0,C 180,E1 -4711.544,E2 -4711.544} C_VEL
LIN {X 0,Y 523.937,Z 333.85,A -85,B 0,C 180,E1 -4714.29,E2 -4714.29} C_VEL
LIN {X 0,Y 523.903,Z 333.836,A -85,B 0,C 180,E1 -4717.133,E2 -4717.133} C_VEL
LIN {X 0,Y 523.96,Z 333.841,A -85,B 0,C 180,E1 -4720.135,E2 -4720.135} C_VEL
LIN {X 0,Y 523.938,Z 333.845,A -85,B 0,C 180,E1 -4722.461,E2 -4722.461} C_VEL
LIN {X 0,Y 523.949,Z 333.833,A -85,B 0,C 180,E1 -4725.31,E2 -4725.31} C_VEL
LIN {X 0,Y 523.966,Z 333.838,A -85,B 0,C 180,E1 -4728.689,E2 -4728.689} C_VEL
LIN {X 0,Y 523.948,Z 333.839,A -85,B 0,C 180,E1 -4731.077,E2 -4731.077} C_VEL
LIN {X 0,Y 523.924,Z 333.848,A -85,B 0,C 180,E1 -4733.829,E2 -4733.829} C_VEL
LIN {X 0,Y 523.94,Z 333.841,A -85,B 0,C 180,E1 -4736.637,E2 -4736.637} C_VEL
LIN {X 0,Y 523.96,Z 333.842,A -85,B 0,C 180,E1 -4739.357,E2 -4739.357} C_VEL
LIN {X 0,Y 523.977,Z 333.843,A -85,B 0,C 180,E1 -4742.282,E2 -4742.282} C_VEL
LIN {X 0,Y 523.953,Z 333.836,A -85,B 0,C 180,E1 -4744.583,E2 -4744.583} C_VEL
LIN {X 0,Y 524.01,Z 333.988,A -85,B 0,C 180,E1 -4745.541,E2 -4745.541} C_VEL
LIN {X 0,Y 525.74,Z 343.558,A -85,B 0,C 180,E1 -4747.192,E2 -4747.192} C_VEL
LIN {X 0,Y 525.131,Z 363.173,A -85,B 0,C 180,E1 -4750.25,E2 -4750.25} C_VEL
LIN {X 0,Y 524.947,Z 372.328,A -85,B 0,C 180,E1 -4751.62,E2 -4751.62} C_VEL
LIN {X 0,Y 527.153,Z 385.142,A -85,B 0,C 180,E1 -4751.901,E2 -4751.901} C_VEL
LIN {X 0,Y 526.459,Z 509.934,A -85,B 0,C 180,E1 -4753.646,E2 -4753.646} C_VEL
LIN {X 0,Y 526.195,Z 524.597,A -85,B 0,C 180,E1 -4754.017,E2 -4754.017} C_VEL
LIN {X 0,Y 525.925,Z 538.848,A -85,B 0,C 180,E1 -4754.549,E2 -4754.549} C_VEL
LIN {X 0,Y 525.606,Z 551.657,A -85,B 0,C 180,E1 -4755.185,E2 -4755.185} C_VEL
LIN {X 0,Y 525.18,Z 564.115,A -85,B 0,C 180,E1 -4755.964,E2 -4755.964} C_VEL
LIN {X 0,Y 524.778,Z 576.662,A -85,B 0,C 180,E1 -4756.94,E2 -4756.94} C_VEL
LIN {X 0,Y 524.447,Z 587.283,A -85,B 0,C 180,E1 -4757.952,E2 -4757.952} C_VEL
LIN {X 0,Y 524.115,Z 597.86,A -85,B 0,C 180,E1 -4759.181,E2 -4759.181} C_VEL
LIN {X 0,Y 523.863,Z 606.18,A -85,B 0,C 180,E1 -4760.347,E2 -4760.347} C_VEL
LIN {X 0,Y 523.663,Z 614.132,A -85,B 0,C 180,E1 -4761.706,E2 -4761.706} C_VEL
LIN {X 0,Y 523.494,Z 620.53,A -85,B 0,C 180,E1 -4763.061,E2 -4763.061} C_VEL
LIN {X 0,Y 523.451,Z 626.204,A -85,B 0,C 180,E1 -4764.608,E2 -4764.608} C_VEL
LIN {X 0,Y 523.418,Z 630.322,A -85,B 0,C 180,E1 -4766.152,E2 -4766.152} C_VEL
LIN {X 0,Y 523.333,Z 633.007,A -85,B 0,C 180,E1 -4767.692,E2 -4767.692} C_VEL
LIN {X 0,Y 523.247,Z 634.335,A -85,B 0,C 180,E1 -4769.231,E2 -4769.231} C_VEL
LIN {X 0,Y 523.247,Z 634.333,A -85,B 0,C 180,E1 -4770.771,E2 -4770.771} C_VEL
LIN {X 0,Y 523.333,Z 633.001,A -85,B 0,C 180,E1 -4772.31,E2 -4772.31} C_VEL
LIN {X 0,Y 523.419,Z 630.313,A -85,B 0,C 180,E1 -4773.85,E2 -4773.85} C_VEL
LIN {X 0,Y 523.453,Z 626.197,A -85,B 0,C 180,E1 -4775.394,E2 -4775.394} C_VEL
LIN {X 0,Y 523.496,Z 620.524,A -85,B 0,C 180,E1 -4776.941,E2 -4776.941} C_VEL
LIN {X 0,Y 523.665,Z 614.121,A -85,B 0,C 180,E1 -4778.296,E2 -4778.296} C_VEL
LIN {X 0,Y 523.863,Z 606.168,A -85,B 0,C 180,E1 -4779.655,E2 -4779.655} C_VEL
LIN {X 0,Y 524.118,Z 597.845,A -85,B 0,C 180,E1 -4780.821,E2 -4780.821} C_VEL
LIN {X 0,Y 524.45,Z 587.082,A -85,B 0,C 180,E1 -4782.069,E2 -4782.069} C_VEL
LIN {X 0,Y 524.755,Z 576.64,A -85,B 0,C 180,E1 -4783.063,E2 -4783.063} C_VEL
LIN {X 0,Y 525.178,Z 564.083,A -85,B 0,C 180,E1 -4784.038,E2 -4784.038} C_VEL
LIN {X 0,Y 525.589,Z 551.62,A -85,B 0,C 180,E1 -4784.818,E2 -4784.818} C_VEL
LIN {X 0,Y 525.936,Z 537.684,A -85,B 0,C 180,E1 -4785.502,E2 -4785.502} C_VEL
LIN {X 0,Y 526.232,Z 523.81,A -85,B 0,C 180,E1 -4786.008,E2 -4786.008} C_VEL
LIN {X 0,Y 526.467,Z 509.845,A -85,B 0,C 180,E1 -4786.356,E2 -4786.356} C_VEL
LIN {X 0,Y 527.177,Z 385.054,A -85,B 0,C 180,E1 -4788.1,E2 -4788.1} C_VEL
LIN {X 0,Y 524.939,Z 372.257,A -85,B 0,C 180,E1 -4788.385,E2 -4788.385} C_VEL
LIN {X 0,Y 525.38,Z 354.006,A -85,B 0,C 180,E1 -4791.173,E2 -4791.173} C_VEL
LIN {X 0,Y 525.658,Z 342.237,A -85,B 0,C 180,E1 -4793.022,E2 -4793.022} C_VEL
LIN {X 0,Y 524.017,Z 333.981,A -85,B 0,C 180,E1 -4794.46,E2 -4794.46} C_VEL
LIN {X 0,Y 523.959,Z 333.843,A -85,B 0,C 180,E1 -4797.133,E2 -4797.133} C_VEL
LIN {X 0,Y 523.947,Z 333.839,A -85,B 0,C 180,E1 -4799.756,E2 -4799.756} C_VEL
LIN {X 0,Y 523.938,Z 333.846,A -85,B 0,C 180,E1 -4802.45,E2 -4802.45} C_VEL
LIN {X 0,Y 523.941,Z 333.843,A -85,B 0,C 180,E1 -4805.226,E2 -4805.226} C_VEL
LIN {X 0,Y 523.921,Z 333.851,A -85,B 0,C 180,E1 -4808.102,E2 -4808.102} C_VEL
LIN {X 0,Y 523.943,Z 333.842,A -85,B 0,C 180,E1 -4811.093,E2 -4811.093} C_VEL
LIN {X 0,Y 523.937,Z 333.846,A -85,B 0,C 180,E1 -4814.229,E2 -4814.229} C_VEL
LIN {X 0,Y 523.926,Z 333.844,A -85,B 0,C 180,E1 -4816.834,E2 -4816.834} C_VEL
LIN {X 0,Y 523.946,Z 333.842,A -85,B 0,C 180,E1 -4818.908,E2 -4818.908} C_VEL
LIN {X 0,Y 523.92,Z 333.851,A -85,B 0,C 180,E1 -4821.899,E2 -4821.899} C_VEL
LIN {X 0,Y 523.929,Z 333.845,A -85,B 0,C 180,E1 -4824.911,E2 -4824.911} C_VEL
LIN {X 0,Y 523.94,Z 333.849,A -85,B 0,C 180,E1 -4827.68,E2 -4827.68} C_VEL
LIN {X 0,Y 523.959,Z 333.843,A -85,B 0,C 180,E1 -4830.677,E2 -4830.677} C_VEL
LIN {X 0,Y 523.991,Z 333.978,A -85,B 0,C 180,E1 -4833.676,E2 -4833.676} C_VEL
LIN {X 0,Y 525.607,Z 342.746,A -85,B 0,C 180,E1 -4834.873,E2 -4834.873} C_VEL
LIN {X 0,Y 525.548,Z 359.345,A -85,B 0,C 180,E1 -4836.974,E2 -4836.974} C_VEL
LIN {X 0,Y 525.243,Z 380.312,A -85,B 0,C 180,E1 -4839.642,E2 -4839.642} C_VEL
LIN {X 0,Y 524.914,Z 399.112,A -85,B 0,C 180,E1 -4842.065,E2 -4842.065} C_VEL
LIN {X 0,Y 524.576,Z 421,A -85,B 0,C 180,E1 -4844.866,E2 -4844.866} C_VEL
LIN {X 0,Y 525.48,Z 427.427,A -85,B 0,C 180,E1 -4845.017,E2 -4845.017} C_VEL
LIN {X 0,Y 525.91,Z 433.025,A -85,B 0,C 180,E1 -4845.112,E2 -4845.112} C_VEL
LIN {X 0,Y 525.397,Z 530.878,A -85,B 0,C 180,E1 -4846.511,E2 -4846.511} C_VEL
LIN {X 0,Y 525.238,Z 544.127,A -85,B 0,C 180,E1 -4846.852,E2 -4846.852} C_VEL
LIN {X 0,Y 524.994,Z 556.655,A -85,B 0,C 180,E1 -4847.337,E2 -4847.337} C_VEL
LIN {X 0,Y 524.751,Z 568.954,A -85,B 0,C 180,E1 -4847.979,E2 -4847.979} C_VEL
LIN {X 0,Y 524.496,Z 579.681,A -85,B 0,C 180,E1 -4848.699,E2 -4848.699} C_VEL
LIN {X 0,Y 524.193,Z 590.101,A -85,B 0,C 180,E1 -4849.572,E2 -4849.572} C_VEL
LIN {X 0,Y 523.981,Z 599.529,A -85,B 0,C 180,E1 -4850.543,E2 -4850.543} C_VEL
LIN {X 0,Y 523.797,Z 607.26,A -85,B 0,C 180,E1 -4851.513,E2 -4851.513} C_VEL
LIN {X 0,Y 523.6,Z 614.802,A -85,B 0,C 180,E1 -4852.674,E2 -4852.674} C_VEL
LIN {X 0,Y 523.506,Z 620.845,A -85,B 0,C 180,E1 -4853.835,E2 -4853.835} C_VEL
LIN {X 0,Y 523.384,Z 625.624,A -85,B 0,C 180,E1 -4854.993,E2 -4854.993} C_VEL
LIN {X 0,Y 523.444,Z 629.281,A -85,B 0,C 180,E1 -4856.151,E2 -4856.151} C_VEL
LIN {X 0,Y 523.368,Z 631.163,A -85,B 0,C 180,E1 -4856.921,E2 -4856.921} C_VEL
LIN {X 0,Y 523.335,Z 632.609,A -85,B 0,C 180,E1 -4857.691,E2 -4857.691} C_VEL
LIN {X 0,Y 523.251,Z 634.241,A -85,B 0,C 180,E1 -4859.23,E2 -4859.23} C_VEL
LIN {X 0,Y 523.247,Z 634.484,A -85,B 0,C 180,E1 -4860,E2 -4860} C_VEL
LIN {X 0,Y 523.25,Z 634.298,A -85,B 0,C 180,E1 -4860.77,E2 -4860.77} C_VEL
LIN {X 0,Y 523.334,Z 632.742,A -85,B 0,C 180,E1 -4862.309,E2 -4862.309} C_VEL
LIN {X 0,Y 523.368,Z 631.369,A -85,B 0,C 180,E1 -4863.079,E2 -4863.079} C_VEL
LIN {X 0,Y 523.425,Z 628.48,A -85,B 0,C 180,E1 -4864.235,E2 -4864.235} C_VEL
LIN {X 0,Y 523.463,Z 624.552,A -85,B 0,C 180,E1 -4865.393,E2 -4865.393} C_VEL
LIN {X 0,Y 523.53,Z 618.846,A -85,B 0,C 180,E1 -4866.673,E2 -4866.673} C_VEL
LIN {X 0,Y 523.691,Z 611.846,A -85,B 0,C 180,E1 -4867.907,E2 -4867.907} C_VEL
LIN {X 0,Y 523.876,Z 603.569,A -85,B 0,C 180,E1 -4869.069,E2 -4869.069} C_VEL
LIN {X 0,Y 524.063,Z 595.053,A -85,B 0,C 180,E1 -4870.04,E2 -4870.04} C_VEL
LIN {X 0,Y 524.373,Z 584.617,A -85,B 0,C 180,E1 -4871.011,E2 -4871.011} C_VEL
LIN {X 0,Y 524.652,Z 574.161,A -85,B 0,C 180,E1 -4871.793,E2 -4871.793} C_VEL
LIN {X 0,Y 524.852,Z 562.751,A -85,B 0,C 180,E1 -4872.47,E2 -4872.47} C_VEL
LIN {X 0,Y 525.155,Z 549.84,A -85,B 0,C 180,E1 -4873.052,E2 -4873.052} C_VEL
LIN {X 0,Y 525.372,Z 536.631,A -85,B 0,C 180,E1 -4873.465,E2 -4873.465} C_VEL
LIN {X 0,Y 525.5,Z 522.489,A -85,B 0,C 180,E1 -4873.732,E2 -4873.732} C_VEL
LIN {X 0,Y 525.896,Z 430.388,A -85,B 0,C 180,E1 -4875.023,E2 -4875.023} C_VEL
LIN {X 0,Y 524.596,Z 421.318,A -85,B 0,C 180,E1 -4875.211,E2 -4875.211} C_VEL
LIN {X 0,Y 524.964,Z 399.081,A -85,B 0,C 180,E1 -4878.098,E2 -4878.098} C_VEL
LIN {X 0,Y 525.463,Z 377.346,A -85,B 0,C 180,E1 -4880.96,E2 -4880.96} C_VEL
LIN {X 0,Y 525.926,Z 355.56,A -85,B 0,C 180,E1 -4883.843,E2 -4883.843} C_VEL
LIN {X 0,Y 526.073,Z 344.569,A -85,B 0,C 180,E1 -4885.309,E2 -4885.309} C_VEL
LIN {X 0,Y 524.007,Z 333.955,A -85,B 0,C 180,E1 -4886.861,E2 -4886.861} C_VEL
LIN {X 0,Y 523.97,Z 333.843,A -85,B 0,C 180,E1 -4887.453,E2 -4887.453} C_VEL
LIN {X 0,Y 523.312,Z 333.927,A -85,B 0,C 180,E1 -4888.095,E2 -4888.095} C_VEL
LIN {X 0,Y 520.43,Z 334.283,A -85,B 0,C 180,E1 -4889.136,E2 -4889.136} C_VEL
LIN {X 0,Y 517.994,Z 334.588,A -85,B 0,C 180,E1 -4889.975,E2 -4889.975} C_VEL
LIN {X 0,Y 516.962,Z 334.719,A -85,B 0,C 180,E1 -4890.623,E2 -4890.623} C_VEL
LIN {X 0,Y 516.886,Z 334.723,A -85,B 0,C 180,E1 -4890.842,E2 -4890.842} C_VEL
LIN {X 0,Y 516.913,Z 334.721,A -85,B 0,C 180,E1 -4893.966,E2 -4893.966} C_VEL
LIN {X 0,Y 516.882,Z 334.724,A -85,B 0,C 180,E1 -4896.746,E2 -4896.746} C_VEL
LIN {X 0,Y 516.887,Z 334.722,A -85,B 0,C 180,E1 -4899.721,E2 -4899.721} C_VEL
LIN {X 0,Y 516.917,Z 334.719,A -85,B 0,C 180,E1 -4901.775,E2 -4901.775} C_VEL
LIN {X 0,Y 516.9,Z 334.711,A -85,B 0,C 180,E1 -4905.007,E2 -4905.007} C_VEL
LIN {X 0,Y 516.918,Z 334.72,A -85,B 0,C 180,E1 -4908.398,E2 -4908.398} C_VEL
LIN {X 0,Y 516.886,Z 334.719,A -85,B 0,C 180,E1 -4911.284,E2 -4911.284} C_VEL
LIN {X 0,Y 516.893,Z 334.722,A -85,B 0,C 180,E1 -4914.221,E2 -4914.221} C_VEL
LIN {X 0,Y 516.9,Z 334.717,A -85,B 0,C 180,E1 -4917.053,E2 -4917.053} C_VEL
LIN {X 0,Y 516.898,Z 334.719,A -85,B 0,C 180,E1 -4919.796,E2 -4919.796} C_VEL
LIN {X 0,Y 516.933,Z 334.72,A -85,B 0,C 180,E1 -4922.467,E2 -4922.467} C_VEL
LIN {X 0,Y 516.973,Z 334.892,A -85,B 0,C 180,E1 -4925.388,E2 -4925.388} C_VEL
LIN {X 0,Y 518.818,Z 344.666,A -85,B 0,C 180,E1 -4927.094,E2 -4927.094} C_VEL
LIN {X 0,Y 518.229,Z 362.874,A -85,B 0,C 180,E1 -4929.974,E2 -4929.974} C_VEL
LIN {X 0,Y 518.006,Z 372.228,A -85,B 0,C 180,E1 -4931.404,E2 -4931.404} C_VEL
LIN {X 0,Y 520.418,Z 385.462,A -85,B 0,C 180,E1 -4931.708,E2 -4931.708} C_VEL
LIN {X 0,Y 519.687,Z 508.892,A -85,B 0,C 180,E1 -4933.45,E2 -4933.45} C_VEL
LIN {X 0,Y 519.41,Z 523.427,A -85,B 0,C 180,E1 -4933.809,E2 -4933.809} C_VEL
LIN {X 0,Y 519.126,Z 536.675,A -85,B 0,C 180,E1 -4934.289,E2 -4934.289} C_VEL
LIN {X 0,Y 518.817,Z 549.066,A -85,B 0,C 180,E1 -4934.884,E2 -4934.884} C_VEL
LIN {X 0,Y 518.345,Z 562.018,A -85,B 0,C 180,E1 -4935.673,E2 -4935.673} C_VEL
LIN {X 0,Y 517.922,Z 573.768,A -85,B 0,C 180,E1 -4936.562,E2 -4936.562} C_VEL
LIN {X 0,Y 517.477,Z 585.294,A -85,B 0,C 180,E1 -4937.628,E2 -4937.628} C_VEL
LIN {X 0,Y 517.18,Z 595.957,A -85,B 0,C 180,E1 -4938.834,E2 -4938.834} C_VEL
LIN {X 0,Y 516.841,Z 604.576,A -85,B 0,C 180,E1 -4940.015,E2 -4940.015} C_VEL
LIN {X 0,Y 516.648,Z 612.875,A -85,B 0,C 180,E1 -4941.393,E2 -4941.393} C_VEL
LIN {X 0,Y 516.456,Z 618.657,A -85,B 0,C 180,E1 -4942.571,E2 -4942.571} C_VEL
LIN {X 0,Y 516.398,Z 624.781,A -85,B 0,C 180,E1 -4944.141,E2 -4944.141} C_VEL
LIN {X 0,Y 516.264,Z 628.33,A -85,B 0,C 180,E1 -4945.314,E2 -4945.314} C_VEL
LIN {X 0,Y 516.325,Z 630.217,A -85,B 0,C 180,E1 -4946.097,E2 -4946.097} C_VEL
LIN {X 0,Y 516.26,Z 632.949,A -85,B 0,C 180,E1 -4947.658,E2 -4947.658} C_VEL
LIN {X 0,Y 516.156,Z 634.274,A -85,B 0,C 180,E1 -4949.219,E2 -4949.219} C_VEL
LIN {X 0,Y 516.153,Z 634.497,A -85,B 0,C 180,E1 -4949.999,E2 -4949.999} C_VEL
LIN {X 0,Y 516.188,Z 633.856,A -85,B 0,C 180,E1 -4951.559,E2 -4951.559} C_VEL
LIN {X 0,Y 516.276,Z 631.879,A -85,B 0,C 180,E1 -4953.12,E2 -4953.12} C_VEL
LIN {X 0,Y 516.325,Z 630.429,A -85,B 0,C 180,E1 -4953.901,E2 -4953.901} C_VEL
LIN {X 0,Y 516.382,Z 626.326,A -85,B 0,C 180,E1 -4955.466,E2 -4955.466} C_VEL
LIN {X 0,Y 516.412,Z 622.223,A -85,B 0,C 180,E1 -4956.656,E2 -4956.656} C_VEL
LIN {X 0,Y 516.5,Z 617.27,A -85,B 0,C 180,E1 -4957.819,E2 -4957.819} C_VEL
LIN {X 0,Y 516.729,Z 610.045,A -85,B 0,C 180,E1 -4959.195,E2 -4959.195} C_VEL
LIN {X 0,Y 516.976,Z 601.154,A -85,B 0,C 180,E1 -4960.574,E2 -4960.574} C_VEL
LIN {X 0,Y 517.317,Z 591.018,A -85,B 0,C 180,E1 -4961.844,E2 -4961.844} C_VEL
LIN {X 0,Y 517.721,Z 580.371,A -85,B 0,C 180,E1 -4962.942,E2 -4962.942} C_VEL
LIN {X 0,Y 518.073,Z 568.731,A -85,B 0,C 180,E1 -4963.932,E2 -4963.932} C_VEL
LIN {X 0,Y 518.555,Z 555.782,A -85,B 0,C 180,E1 -4964.821,E2 -4964.821} C_VEL
LIN {X 0,Y 518.991,Z 542.07,A -85,B 0,C 180,E1 -4965.562,E2 -4965.562} C_VEL
LIN {X 0,Y 519.279,Z 529.251,A -85,B 0,C 180,E1 -4966.09,E2 -4966.09} C_VEL
LIN {X 0,Y 519.601,Z 515.378,A -85,B 0,C 180,E1 -4966.5,E2 -4966.5} C_VEL
LIN {X 0,Y 519.758,Z 500.513,A -85,B 0,C 180,E1 -4966.773,E2 -4966.773} C_VEL
LIN {X 0,Y 520.422,Z 385.113,A -85,B 0,C 180,E1 -4968.387,E2 -4968.387} C_VEL
LIN {X 0,Y 518,Z 372.266,A -85,B 0,C 180,E1 -4968.684,E2 -4968.684} C_VEL
LIN {X 0,Y 518.431,Z 355.611,A -85,B 0,C 180,E1 -4971.26,E2 -4971.26} C_VEL
LIN {X 0,Y 518.762,Z 343.837,A -85,B 0,C 180,E1 -4973.133,E2 -4973.133} C_VEL
LIN {X 0,Y 516.953,Z 334.816,A -85,B 0,C 180,E1 -4974.735,E2 -4974.735} C_VEL
LIN {X 0,Y 516.929,Z 334.719,A -85,B 0,C 180,E1 -4977.531,E2 -4977.531} C_VEL
LIN {X 0,Y 516.9,Z 334.717,A -85,B 0,C 180,E1 -4980.202,E2 -4980.202} C_VEL
LIN {X 0,Y 516.896,Z 334.718,A -85,B 0,C 180,E1 -4982.945,E2 -4982.945} C_VEL
LIN {X 0,Y 516.887,Z 334.723,A -85,B 0,C 180,E1 -4985.777,E2 -4985.777} C_VEL
LIN {X 0,Y 516.915,Z 334.715,A -85,B 0,C 180,E1 -4989.197,E2 -4989.197} C_VEL
LIN {X 0,Y 516.913,Z 334.721,A -85,B 0,C 180,E1 -4991.773,E2 -4991.773} C_VEL
LIN {X 0,Y 516.916,Z 334.709,A -85,B 0,C 180,E1 -4995.009,E2 -4995.009} C_VEL
LIN {X 0,Y 516.923,Z 334.717,A -85,B 0,C 180,E1 -4998.396,E2 -4998.396} C_VEL
LIN {X 0,Y 516.899,Z 334.716,A -85,B 0,C 180,E1 -5001.286,E2 -5001.286} C_VEL
LIN {X 0,Y 516.883,Z 334.721,A -85,B 0,C 180,E1 -5004.22,E2 -5004.22} C_VEL
LIN {X 0,Y 516.89,Z 334.721,A -85,B 0,C 180,E1 -5007.053,E2 -5007.053} C_VEL
LIN {X 0,Y 516.893,Z 334.71,A -85,B 0,C 180,E1 -5009.796,E2 -5009.796} C_VEL
LIN {X 0,Y 516.921,Z 334.707,A -85,B 0,C 180,E1 -5012.467,E2 -5012.467} C_VEL
LIN {X 0,Y 516.905,Z 334.719,A -85,B 0,C 180,E1 -5015.071,E2 -5015.071} C_VEL
LIN {X 0,Y 516.903,Z 334.72,A -85,B 0,C 180,E1 -5017.623,E2 -5017.623} C_VEL
LIN {X 0,Y 516.923,Z 334.715,A -85,B 0,C 180,E1 -5020.129,E2 -5020.129} C_VEL
LIN {X 0,Y 516.922,Z 334.715,A -85,B 0,C 180,E1 -5022.596,E2 -5022.596} C_VEL
LIN {X 0,Y 516.94,Z 334.712,A -85,B 0,C 180,E1 -5025.03,E2 -5025.03} C_VEL
LIN {X 0,Y 516.993,Z 334.705,A -85,B 0,C 180,E1 -5028.234,E2 -5028.234} C_VEL
LIN {X 0,Y 516.964,Z 334.714,A -85,B 0,C 180,E1 -5031.4,E2 -5031.4} C_VEL
LIN {X 0,Y 517.035,Z 334.702,A -85,B 0,C 180,E1 -5034.54,E2 -5034.54} C_VEL
LIN {X 0,Y 517.075,Z 334.695,A -85,B 0,C 180,E1 -5037.663,E2 -5037.663} C_VEL
LIN {X 0,Y 517.088,Z 334.7,A -85,B 0,C 180,E1 -5040.779,E2 -5040.779} C_VEL
LIN {X 0,Y 517.009,Z 334.706,A -85,B 0,C 180,E1 -5043.117,E2 -5043.117} C_VEL
LIN {X 0,Y 517.001,Z 334.706,A -85,B 0,C 180,E1 -5046.243,E2 -5046.243} C_VEL
LIN {X 0,Y 516.95,Z 334.707,A -85,B 0,C 180,E1 -5049.389,E2 -5049.389} C_VEL
LIN {X 0,Y 516.972,Z 334.707,A -85,B 0,C 180,E1 -5051.824,E2 -5051.824} C_VEL
LIN {X 0,Y 516.936,Z 334.71,A -85,B 0,C 180,E1 -5055.148,E2 -5055.148} C_VEL
LIN {X 0,Y 516.916,Z 334.718,A -85,B 0,C 180,E1 -5058.223,E2 -5058.223} C_VEL
LIN {X 0,Y 516.905,Z 334.719,A -85,B 0,C 180,E1 -5060.702,E2 -5060.702} C_VEL
LIN {X 0,Y 516.882,Z 334.721,A -85,B 0,C 180,E1 -5063.223,E2 -5063.223} C_VEL
LIN {X 0,Y 516.935,Z 334.716,A -85,B 0,C 180,E1 -5066.197,E2 -5066.197} C_VEL
LIN {X 0,Y 516.913,Z 334.701,A -85,B 0,C 180,E1 -5069.305,E2 -5069.305} C_VEL
LIN {X 0,Y 516.892,Z 334.726,A -85,B 0,C 180,E1 -5072.545,E2 -5072.545} C_VEL
LIN {X 0,Y 516.875,Z 334.719,A -85,B 0,C 180,E1 -5075.333,E2 -5075.333} C_VEL
LIN {X 0,Y 516.873,Z 334.714,A -85,B 0,C 180,E1 -5077.944,E2 -5077.944} C_VEL
LIN {X 0,Y 516.901,Z 334.721,A -85,B 0,C 180,E1 -5080.74,E2 -5080.74} C_VEL
LIN {X 0,Y 516.877,Z 334.724,A -85,B 0,C 180,E1 -5083.904,E2 -5083.904} C_VEL
LIN {X 0,Y 516.875,Z 334.723,A -85,B 0,C 180,E1 -5086.108,E2 -5086.108} C_VEL
LIN {X 0,Y 516.898,Z 334.717,A -85,B 0,C 180,E1 -5089.261,E2 -5089.261} C_VEL
LIN {X 0,Y 516.877,Z 334.73,A -85,B 0,C 180,E1 -5092.058,E2 -5092.058} C_VEL
LIN {X 0,Y 516.892,Z 334.719,A -85,B 0,C 180,E1 -5095.177,E2 -5095.177} C_VEL
LIN {X 0,Y 516.88,Z 334.727,A -85,B 0,C 180,E1 -5097.977,E2 -5097.977} C_VEL
LIN {X 0,Y 516.933,Z 334.702,A -85,B 0,C 180,E1 -5100.698,E2 -5100.698} C_VEL
LIN {X 0,Y 516.942,Z 334.71,A -85,B 0,C 180,E1 -5103.804,E2 -5103.804} C_VEL
LIN {X 0,Y 516.935,Z 334.814,A -85,B 0,C 180,E1 -5105.307,E2 -5105.307} C_VEL
LIN {X 0,Y 518.478,Z 342.251,A -85,B 0,C 180,E1 -5106.643,E2 -5106.643} C_VEL
LIN {X 0,Y 518.848,Z 344.886,A -85,B 0,C 180,E1 -5107.086,E2 -5107.086} C_VEL
LIN {X 0,Y 518.193,Z 364.48,A -85,B 0,C 180,E1 -5110.181,E2 -5110.181} C_VEL
LIN {X 0,Y 517.999,Z 372.226,A -85,B 0,C 180,E1 -5111.358,E2 -5111.358} C_VEL
LIN {X 0,Y 520.416,Z 385.758,A -85,B 0,C 180,E1 -5111.667,E2 -5111.667} C_VEL
LIN {X 0,Y 519.647,Z 509.934,A -85,B 0,C 180,E1 -5113.425,E2 -5113.425} C_VEL
LIN {X 0,Y 519.386,Z 524.552,A -85,B 0,C 180,E1 -5113.801,E2 -5113.801} C_VEL
LIN {X 0,Y 519.088,Z 538.848,A -85,B 0,C 180,E1 -5114.341,E2 -5114.341} C_VEL
LIN {X 0,Y 518.719,Z 551.657,A -85,B 0,C 180,E1 -5114.983,E2 -5114.983} C_VEL
LIN {X 0,Y 518.287,Z 564.115,A -85,B 0,C 180,E1 -5115.773,E2 -5115.773} C_VEL
LIN {X 0,Y 517.826,Z 576.662,A -85,B 0,C 180,E1 -5116.761,E2 -5116.761} C_VEL
LIN {X 0,Y 517.452,Z 587.668,A -85,B 0,C 180,E1 -5117.829,E2 -5117.829} C_VEL
LIN {X 0,Y 517.107,Z 597.86,A -85,B 0,C 180,E1 -5119.032,E2 -5119.032} C_VEL
LIN {X 0,Y 516.827,Z 606.18,A -85,B 0,C 180,E1 -5120.214,E2 -5120.214} C_VEL
LIN {X 0,Y 516.598,Z 614.132,A -85,B 0,C 180,E1 -5121.592,E2 -5121.592} C_VEL
LIN {X 0,Y 516.405,Z 620.53,A -85,B 0,C 180,E1 -5122.966,E2 -5122.966} C_VEL
LIN {X 0,Y 516.407,Z 624.962,A -85,B 0,C 180,E1 -5124.143,E2 -5124.143} C_VEL
LIN {X 0,Y 516.264,Z 628.449,A -85,B 0,C 180,E1 -5125.316,E2 -5125.316} C_VEL
LIN {X 0,Y 516.324,Z 630.322,A -85,B 0,C 180,E1 -5126.099,E2 -5126.099} C_VEL
LIN {X 0,Y 516.259,Z 633.007,A -85,B 0,C 180,E1 -5127.66,E2 -5127.66} C_VEL
LIN {X 0,Y 516.157,Z 634.335,A -85,B 0,C 180,E1 -5129.221,E2 -5129.221} C_VEL
LIN {X 0,Y 516.157,Z 634.333,A -85,B 0,C 180,E1 -5130.781,E2 -5130.781} C_VEL
LIN {X 0,Y 516.259,Z 633.001,A -85,B 0,C 180,E1 -5132.342,E2 -5132.342} C_VEL
LIN {X 0,Y 516.325,Z 630.313,A -85,B 0,C 180,E1 -5133.903,E2 -5133.903} C_VEL
LIN {X 0,Y 516.389,Z 626.197,A -85,B 0,C 180,E1 -5135.468,E2 -5135.468} C_VEL
LIN {X 0,Y 516.407,Z 620.524,A -85,B 0,C 180,E1 -5137.036,E2 -5137.036} C_VEL
LIN {X 0,Y 516.6,Z 614.121,A -85,B 0,C 180,E1 -5138.41,E2 -5138.41} C_VEL
LIN {X 0,Y 516.827,Z 606.168,A -85,B 0,C 180,E1 -5139.788,E2 -5139.788} C_VEL
LIN {X 0,Y 517.11,Z 597.845,A -85,B 0,C 180,E1 -5140.97,E2 -5140.97} C_VEL
LIN {X 0,Y 517.459,Z 587.425,A -85,B 0,C 180,E1 -5142.198,E2 -5142.198} C_VEL
LIN {X 0,Y 517.841,Z 576.64,A -85,B 0,C 180,E1 -5143.24,E2 -5143.24} C_VEL
LIN {X 0,Y 518.27,Z 564.083,A -85,B 0,C 180,E1 -5144.229,E2 -5144.229} C_VEL
LIN {X 0,Y 518.729,Z 551.62,A -85,B 0,C 180,E1 -5145.018,E2 -5145.018} C_VEL
LIN {X 0,Y 519.068,Z 538.813,A -85,B 0,C 180,E1 -5145.662,E2 -5145.662} C_VEL
LIN {X 0,Y 519.394,Z 524.829,A -85,B 0,C 180,E1 -5146.19,E2 -5146.19} C_VEL
LIN {X 0,Y 519.661,Z 510.985,A -85,B 0,C 180,E1 -5146.551,E2 -5146.551} C_VEL
LIN {X 0,Y 519.849,Z 484.664,A -85,B 0,C 180,E1 -5146.949,E2 -5146.949} C_VEL
LIN {X 0,Y 520.354,Z 384.896,A -85,B 0,C 180,E1 -5148.348,E2 -5148.348} C_VEL
LIN {X 0,Y 518.013,Z 372.263,A -85,B 0,C 180,E1 -5148.638,E2 -5148.638} C_VEL
LIN {X 0,Y 518.527,Z 354.006,A -85,B 0,C 180,E1 -5151.467,E2 -5151.467} C_VEL
LIN {X 0,Y 518.715,Z 343.545,A -85,B 0,C 180,E1 -5153.137,E2 -5153.137} C_VEL
LIN {X 0,Y 517,Z 335.045,A -85,B 0,C 180,E1 -5154.616,E2 -5154.616} C_VEL
LIN {X 0,Y 516.932,Z 334.715,A -85,B 0,C 180,E1 -5154.928,E2 -5154.928} C_VEL
LIN {X 0,Y 516.932,Z 334.715,A -85,B 0,C 180,E1 -5157.906,E2 -5157.906} C_VEL
LIN {X 0,Y 516.897,Z 334.724,A -85,B 0,C 180,E1 -5160.204,E2 -5160.204} C_VEL
LIN {X 0,Y 516.9,Z 334.719,A -85,B 0,C 180,E1 -5162.947,E2 -5162.947} C_VEL
LIN {X 0,Y 516.896,Z 334.726,A -85,B 0,C 180,E1 -5165.779,E2 -5165.779} C_VEL
LIN {X 0,Y 516.885,Z 334.722,A -85,B 0,C 180,E1 -5168.716,E2 -5168.716} C_VEL
LIN {X 0,Y 516.916,Z 334.722,A -85,B 0,C 180,E1 -5171.776,E2 -5171.776} C_VEL
LIN {X 0,Y 516.899,Z 334.719,A -85,B 0,C 180,E1 -5175.007,E2 -5175.007} C_VEL
LIN {X 0,Y 516.92,Z 334.719,A -85,B 0,C 180,E1 -5178.399,E2 -5178.399} C_VEL
LIN {X 0,Y 516.885,Z 334.724,A -85,B 0,C 180,E1 -5181.284,E2 -5181.284} C_VEL
LIN {X 0,Y 516.875,Z 334.725,A -85,B 0,C 180,E1 -5184.22,E2 -5184.22} C_VEL
LIN {X 0,Y 516.899,Z 334.722,A -85,B 0,C 180,E1 -5187.053,E2 -5187.053} C_VEL
LIN {X 0,Y 516.897,Z 334.727,A -85,B 0,C 180,E1 -5189.797,E2 -5189.797} C_VEL
LIN {X 0,Y 516.934,Z 334.72,A -85,B 0,C 180,E1 -5192.468,E2 -5192.468} C_VEL
LIN {X 0,Y 516.991,Z 334.927,A -85,B 0,C 180,E1 -5193.521,E2 -5193.521} C_VEL
LIN {X 0,Y 518.809,Z 345.475,A -85,B 0,C 180,E1 -5194.955,E2 -5194.955} C_VEL
LIN {X 0,Y 518.48,Z 368.593,A -85,B 0,C 180,E1 -5197.905,E2 -5197.905} C_VEL
LIN {X 0,Y 518.103,Z 389.379,A -85,B 0,C 180,E1 -5200.589,E2 -5200.589} C_VEL
LIN {X 0,Y 517.772,Z 411.376,A -85,B 0,C 180,E1 -5203.439,E2 -5203.439} C_VEL
LIN {X 0,Y 517.6,Z 421.215,A -85,B 0,C 180,E1 -5204.681,E2 -5204.681} C_VEL
LIN {X 0,Y 519.063,Z 431.7,A -85,B 0,C 180,E1 -5204.897,E2 -5204.897} C_VEL
LIN {X 0,Y 518.464,Z 530.867,A -85,B 0,C 180,E1 -5206.352,E2 -5206.352} C_VEL
LIN {X 0,Y 518.317,Z 543.307,A -85,B 0,C 180,E1 -5206.673,E2 -5206.673} C_VEL
LIN {X 0,Y 518.025,Z 556.097,A -85,B 0,C 180,E1 -5207.164,E2 -5207.164} C_VEL
LIN {X 0,Y 517.757,Z 568.951,A -85,B 0,C 180,E1 -5207.84,E2 -5207.84} C_VEL
LIN {X 0,Y 517.471,Z 580.605,A -85,B 0,C 180,E1 -5208.642,E2 -5208.642} C_VEL
LIN {X 0,Y 517.137,Z 590.885,A -85,B 0,C 180,E1 -5209.527,E2 -5209.527} C_VEL
LIN {X 0,Y 516.947,Z 599.322,A -85,B 0,C 180,E1 -5210.413,E2 -5210.413} C_VEL
LIN {X 0,Y 516.749,Z 607.096,A -85,B 0,C 180,E1 -5211.396,E2 -5211.396} C_VEL
LIN {X 0,Y 516.524,Z 614.686,A -85,B 0,C 180,E1 -5212.573,E2 -5212.573} C_VEL
LIN {X 0,Y 516.407,Z 620.758,A -85,B 0,C 180,E1 -5213.75,E2 -5213.75} C_VEL
LIN {X 0,Y 516.314,Z 625.562,A -85,B 0,C 180,E1 -5214.924,E2 -5214.924} C_VEL
LIN {X 0,Y 516.353,Z 629.239,A -85,B 0,C 180,E1 -5216.098,E2 -5216.098} C_VEL
LIN {X 0,Y 516.283,Z 631.131,A -85,B 0,C 180,E1 -5216.879,E2 -5216.879} C_VEL
LIN {X 0,Y 516.261,Z 632.586,A -85,B 0,C 180,E1 -5217.659,E2 -5217.659} C_VEL
LIN {X 0,Y 516.161,Z 634.226,A -85,B 0,C 180,E1 -5219.22,E2 -5219.22} C_VEL
LIN {X 0,Y 516.154,Z 634.47,A -85,B 0,C 180,E1 -5220,E2 -5220} C_VEL
LIN {X 0,Y 516.16,Z 634.283,A -85,B 0,C 180,E1 -5220.78,E2 -5220.78} C_VEL
LIN {X 0,Y 516.261,Z 632.718,A -85,B 0,C 180,E1 -5222.341,E2 -5222.341} C_VEL
LIN {X 0,Y 516.283,Z 631.338,A -85,B 0,C 180,E1 -5223.121,E2 -5223.121} C_VEL
LIN {X 0,Y 516.331,Z 628.435,A -85,B 0,C 180,E1 -5224.293,E2 -5224.293} C_VEL
LIN {X 0,Y 516.4,Z 624.487,A -85,B 0,C 180,E1 -5225.467,E2 -5225.467} C_VEL
LIN {X 0,Y 516.475,Z 618.621,A -85,B 0,C 180,E1 -5226.792,E2 -5226.792} C_VEL
LIN {X 0,Y 516.639,Z 611.724,A -85,B 0,C 180,E1 -5228.015,E2 -5228.015} C_VEL
LIN {X 0,Y 516.831,Z 603.404,A -85,B 0,C 180,E1 -5229.194,E2 -5229.194} C_VEL
LIN {X 0,Y 517.036,Z 594.85,A -85,B 0,C 180,E1 -5230.178,E2 -5230.178} C_VEL
LIN {X 0,Y 517.368,Z 584.366,A -85,B 0,C 180,E1 -5231.162,E2 -5231.162} C_VEL
LIN {X 0,Y 517.658,Z 573.874,A -85,B 0,C 180,E1 -5231.952,E2 -5231.952} C_VEL
LIN {X 0,Y 517.908,Z 562.343,A -85,B 0,C 180,E1 -5232.64,E2 -5232.64} C_VEL
LIN {X 0,Y 518.211,Z 549.302,A -85,B 0,C 180,E1 -5233.23,E2 -5233.23} C_VEL
LIN {X 0,Y 518.452,Z 535.825,A -85,B 0,C 180,E1 -5233.648,E2 -5233.648} C_VEL
LIN {X 0,Y 518.578,Z 522.867,A -85,B 0,C 180,E1 -5233.894,E2 -5233.894} C_VEL
LIN {X 0,Y 519.062,Z 431.151,A -85,B 0,C 180,E1 -5235.21,E2 -5235.21} C_VEL
LIN {X 0,Y 517.615,Z 421.278,A -85,B 0,C 180,E1 -5235.416,E2 -5235.416} C_VEL
LIN {X 0,Y 518.115,Z 397.399,A -85,B 0,C 180,E1 -5238.547,E2 -5238.547} C_VEL
LIN {X 0,Y 518.61,Z 373.931,A -85,B 0,C 180,E1 -5241.671,E2 -5241.671} C_VEL
LIN {X 0,Y 519.118,Z 353.603,A -85,B 0,C 180,E1 -5244.388,E2 -5244.388} C_VEL
LIN {X 0,Y 519.16,Z 345.867,A -85,B 0,C 180,E1 -5245.434,E2 -5245.434} C_VEL
LIN {X 0,Y 516.968,Z 334.829,A -85,B 0,C 180,E1 -5247.065,E2 -5247.065} C_VEL
LIN {X 0,Y 516.897,Z 334.726,A -85,B 0,C 180,E1 -5250.204,E2 -5250.204} C_VEL
LIN {X 0,Y 516.886,Z 334.723,A -85,B 0,C 180,E1 -5250.842,E2 -5250.842} C_VEL
LIN {X 0,Y 516.244,Z 334.804,A -85,B 0,C 180,E1 -5251.493,E2 -5251.493} C_VEL
LIN {X 0,Y 513.412,Z 335.161,A -85,B 0,C 180,E1 -5252.549,E2 -5252.549} C_VEL
LIN {X 0,Y 510.996,Z 335.46,A -85,B 0,C 180,E1 -5253.4,E2 -5253.4} C_VEL
LIN {X 0,Y 509.948,Z 335.591,A -85,B 0,C 180,E1 -5254.057,E2 -5254.057} C_VEL
LIN {X 0,Y 509.857,Z 335.603,A -85,B 0,C 180,E1 -5254.279,E2 -5254.279} C_VEL
LIN {X 0,Y 509.822,Z 335.6,A -85,B 0,C 180,E1 -5257.341,E2 -5257.341} C_VEL
LIN {X 0,Y 509.843,Z 335.604,A -85,B 0,C 180,E1 -5260.382,E2 -5260.382} C_VEL
LIN {X 0,Y 509.827,Z 335.597,A -85,B 0,C 180,E1 -5263.062,E2 -5263.062} C_VEL
LIN {X 0,Y 509.828,Z 335.595,A -85,B 0,C 180,E1 -5265.793,E2 -5265.793} C_VEL
LIN {X 0,Y 509.86,Z 335.597,A -85,B 0,C 180,E1 -5268.574,E2 -5268.574} C_VEL
LIN {X 0,Y 509.856,Z 335.599,A -85,B 0,C 180,E1 -5271.786,E2 -5271.786} C_VEL
LIN {X 0,Y 509.848,Z 335.598,A -85,B 0,C 180,E1 -5274.623,E2 -5274.623} C_VEL
LIN {X 0,Y 509.867,Z 335.596,A -85,B 0,C 180,E1 -5277.48,E2 -5277.48} C_VEL
LIN {X 0,Y 509.864,Z 335.586,A -85,B 0,C 180,E1 -5280.273,E2 -5280.273} C_VEL
LIN {X 0,Y 509.891,Z 335.596,A -85,B 0,C 180,E1 -5282.944,E2 -5282.944} C_VEL
LIN {X 0,Y 509.945,Z 335.745,A -85,B 0,C 180,E1 -5285.164,E2 -5285.164} C_VEL
LIN {X 0,Y 511.921,Z 346.425,A -85,B 0,C 180,E1 -5287.054,E2 -5287.054} C_VEL
LIN {X 0,Y 511.288,Z 364.185,A -85,B 0,C 180,E1 -5289.9,E2 -5289.9} C_VEL
LIN {X 0,Y 511.093,Z 372.262,A -85,B 0,C 180,E1 -5291.145,E2 -5291.145} C_VEL
LIN {X 0,Y 513.672,Z 386.478,A -85,B 0,C 180,E1 -5291.473,E2 -5291.473} C_VEL
LIN {X 0,Y 512.889,Z 508.927,A -85,B 0,C 180,E1 -5293.224,E2 -5293.224} C_VEL
LIN {X 0,Y 512.617,Z 523.289,A -85,B 0,C 180,E1 -5293.583,E2 -5293.583} C_VEL
LIN {X 0,Y 512.299,Z 536.69,A -85,B 0,C 180,E1 -5294.075,E2 -5294.075} C_VEL
LIN {X 0,Y 511.962,Z 549.077,A -85,B 0,C 180,E1 -5294.676,E2 -5294.676} C_VEL
LIN {X 0,Y 511.441,Z 562.027,A -85,B 0,C 180,E1 -5295.475,E2 -5295.475} C_VEL
LIN {X 0,Y 510.987,Z 573.773,A -85,B 0,C 180,E1 -5296.376,E2 -5296.376} C_VEL
LIN {X 0,Y 510.501,Z 585.474,A -85,B 0,C 180,E1 -5297.474,E2 -5297.474} C_VEL
LIN {X 0,Y 510.191,Z 595.962,A -85,B 0,C 180,E1 -5298.679,E2 -5298.679} C_VEL
LIN {X 0,Y 509.815,Z 604.599,A -85,B 0,C 180,E1 -5299.876,E2 -5299.876} C_VEL
LIN {X 0,Y 509.586,Z 612.882,A -85,B 0,C 180,E1 -5301.273,E2 -5301.273} C_VEL
LIN {X 0,Y 509.385,Z 618.656,A -85,B 0,C 180,E1 -5302.468,E2 -5302.468} C_VEL
LIN {X 0,Y 509.309,Z 623.41,A -85,B 0,C 180,E1 -5303.661,E2 -5303.661} C_VEL
LIN {X 0,Y 509.238,Z 627.262,A -85,B 0,C 180,E1 -5304.852,E2 -5304.852} C_VEL
LIN {X 0,Y 509.22,Z 630.215,A -85,B 0,C 180,E1 -5306.042,E2 -5306.042} C_VEL
LIN {X 0,Y 509.16,Z 632.946,A -85,B 0,C 180,E1 -5307.626,E2 -5307.626} C_VEL
LIN {X 0,Y 509.07,Z 634.299,A -85,B 0,C 180,E1 -5309.208,E2 -5309.208} C_VEL
LIN {X 0,Y 509.071,Z 634.33,A -85,B 0,C 180,E1 -5310.79,E2 -5310.79} C_VEL
LIN {X 0,Y 509.159,Z 633.066,A -85,B 0,C 180,E1 -5312.372,E2 -5312.372} C_VEL
LIN {X 0,Y 509.219,Z 630.425,A -85,B 0,C 180,E1 -5313.956,E2 -5313.956} C_VEL
LIN {X 0,Y 509.315,Z 626.337,A -85,B 0,C 180,E1 -5315.542,E2 -5315.542} C_VEL
LIN {X 0,Y 509.338,Z 622.453,A -85,B 0,C 180,E1 -5316.695,E2 -5316.695} C_VEL
LIN {X 0,Y 509.45,Z 617.264,A -85,B 0,C 180,E1 -5317.928,E2 -5317.928} C_VEL
LIN {X 0,Y 509.676,Z 610.059,A -85,B 0,C 180,E1 -5319.323,E2 -5319.323} C_VEL
LIN {X 0,Y 509.897,Z 602.512,A -85,B 0,C 180,E1 -5320.522,E2 -5320.522} C_VEL
LIN {X 0,Y 510.271,Z 593.452,A -85,B 0,C 180,E1 -5321.72,E2 -5321.72} C_VEL
LIN {X 0,Y 510.592,Z 584.429,A -85,B 0,C 180,E1 -5322.721,E2 -5322.721} C_VEL
LIN {X 0,Y 510.995,Z 573.665,A -85,B 0,C 180,E1 -5323.723,E2 -5323.723} C_VEL
LIN {X 0,Y 511.463,Z 561.896,A -85,B 0,C 180,E1 -5324.624,E2 -5324.624} C_VEL
LIN {X 0,Y 511.883,Z 548.903,A -85,B 0,C 180,E1 -5325.426,E2 -5325.426} C_VEL
LIN {X 0,Y 512.382,Z 535.033,A -85,B 0,C 180,E1 -5326.085,E2 -5326.085} C_VEL
LIN {X 0,Y 512.68,Z 520.845,A -85,B 0,C 180,E1 -5326.578,E2 -5326.578} C_VEL
LIN {X 0,Y 512.899,Z 506.828,A -85,B 0,C 180,E1 -5326.902,E2 -5326.902} C_VEL
LIN {X 0,Y 513.644,Z 385.747,A -85,B 0,C 180,E1 -5328.629,E2 -5328.629} C_VEL
LIN {X 0,Y 511.103,Z 372.502,A -85,B 0,C 180,E1 -5328.932,E2 -5328.932} C_VEL
LIN {X 0,Y 511.106,Z 369.993,A -85,B 0,C 180,E1 -5329.268,E2 -5329.268} C_VEL
LIN {X 0,Y 511.694,Z 352.989,A -85,B 0,C 180,E1 -5331.978,E2 -5331.978} C_VEL
LIN {X 0,Y 511.87,Z 345.348,A -85,B 0,C 180,E1 -5333.215,E2 -5333.215} C_VEL
LIN {X 0,Y 509.919,Z 335.712,A -85,B 0,C 180,E1 -5334.944,E2 -5334.944} C_VEL
LIN {X 0,Y 509.894,Z 335.593,A -85,B 0,C 180,E1 -5337.944,E2 -5337.944} C_VEL
LIN {X 0,Y 509.848,Z 335.601,A -85,B 0,C 180,E1 -5340.664,E2 -5340.664} C_VEL
LIN {X 0,Y 509.861,Z 335.595,A -85,B 0,C 180,E1 -5343.459,E2 -5343.459} C_VEL
LIN {X 0,Y 509.832,Z 335.603,A -85,B 0,C 180,E1 -5346.351,E2 -5346.351} C_VEL
LIN {X 0,Y 509.861,Z 335.596,A -85,B 0,C 180,E1 -5349.474,E2 -5349.474} C_VEL
LIN {X 0,Y 509.861,Z 335.597,A -85,B 0,C 180,E1 -5352.485,E2 -5352.485} C_VEL
LIN {X 0,Y 509.85,Z 335.59,A -85,B 0,C 180,E1 -5355.331,E2 -5355.331} C_VEL
LIN {X 0,Y 509.864,Z 335.595,A -85,B 0,C 180,E1 -5358.575,E2 -5358.575} C_VEL
LIN {X 0,Y 509.848,Z 335.59,A -85,B 0,C 180,E1 -5361.785,E2 -5361.785} C_VEL
LIN {X 0,Y 509.838,Z 335.596,A -85,B 0,C 180,E1 -5364.622,E2 -5364.622} C_VEL
LIN {X 0,Y 509.858,Z 335.602,A -85,B 0,C 180,E1 -5367.48,E2 -5367.48} C_VEL
LIN {X 0,Y 509.873,Z 335.578,A -85,B 0,C 180,E1 -5370.268,E2 -5370.268} C_VEL
LIN {X 0,Y 509.878,Z 335.585,A -85,B 0,C 180,E1 -5372.944,E2 -5372.944} C_VEL
LIN {X 0,Y 509.866,Z 335.602,A -85,B 0,C 180,E1 -5375.574,E2 -5375.574} C_VEL
LIN {X 0,Y 509.839,Z 335.594,A -85,B 0,C 180,E1 -5378.149,E2 -5378.149} C_VEL
LIN {X 0,Y 509.856,Z 335.595,A -85,B 0,C 180,E1 -5380.681,E2 -5380.681} C_VEL
LIN {X 0,Y 509.878,Z 335.598,A -85,B 0,C 180,E1 -5383.174,E2 -5383.174} C_VEL
LIN {X 0,Y 509.864,Z 335.597,A -85,B 0,C 180,E1 -5385.634,E2 -5385.634} C_VEL
LIN {X 0,Y 509.92,Z 335.59,A -85,B 0,C 180,E1 -5388.875,E2 -5388.875} C_VEL
LIN {X 0,Y 509.942,Z 335.583,A -85,B 0,C 180,E1 -5392.078,E2 -5392.078} C_VEL
LIN {X 0,Y 509.985,Z 335.58,A -85,B 0,C 180,E1 -5394.464,E2 -5394.464} C_VEL
LIN {X 0,Y 510.046,Z 335.571,A -85,B 0,C 180,E1 -5397.631,E2 -5397.631} C_VEL
LIN {X 0,Y 510.057,Z 335.576,A -85,B 0,C 180,E1 -5400.789,E2 -5400.789} C_VEL
LIN {X 0,Y 509.952,Z 335.584,A -85,B 0,C 180,E1 -5403.16,E2 -5403.16} C_VEL
LIN {X 0,Y 509.969,Z 335.583,A -85,B 0,C 180,E1 -5406.33,E2 -5406.33} C_VEL
LIN {X 0,Y 509.91,Z 335.592,A -85,B 0,C 180,E1 -5408.72,E2 -5408.72} C_VEL
LIN {X 0,Y 509.94,Z 335.584,A -85,B 0,C 180,E1 -5411.931,E2 -5411.931} C_VEL
LIN {X 0,Y 509.882,Z 335.588,A -85,B 0,C 180,E1 -5415.242,E2 -5415.242} C_VEL
LIN {X 0,Y 509.878,Z 335.592,A -85,B 0,C 180,E1 -5418.002,E2 -5418.002} C_VEL
LIN {X 0,Y 509.847,Z 335.595,A -85,B 0,C 180,E1 -5421.002,E2 -5421.002} C_VEL
LIN {X 0,Y 509.841,Z 335.597,A -85,B 0,C 180,E1 -5423.563,E2 -5423.563} C_VEL
LIN {X 0,Y 509.904,Z 335.592,A -85,B 0,C 180,E1 -5426.38,E2 -5426.38} C_VEL
LIN {X 0,Y 509.868,Z 335.58,A -85,B 0,C 180,E1 -5428.845,E2 -5428.845} C_VEL
LIN {X 0,Y 509.816,Z 335.596,A -85,B 0,C 180,E1 -5431.59,E2 -5431.59} C_VEL
LIN {X 0,Y 509.846,Z 335.603,A -85,B 0,C 180,E1 -5434.414,E2 -5434.414} C_VEL
LIN {X 0,Y 509.811,Z 335.59,A -85,B 0,C 180,E1 -5437.341,E2 -5437.341} C_VEL
LIN {X 0,Y 509.855,Z 335.602,A -85,B 0,C 180,E1 -5440.381,E2 -5440.381} C_VEL
LIN {X 0,Y 509.834,Z 335.596,A -85,B 0,C 180,E1 -5443.065,E2 -5443.065} C_VEL
LIN {X 0,Y 509.823,Z 335.596,A -85,B 0,C 180,E1 -5445.793,E2 -5445.793} C_VEL
LIN {X 0,Y 509.859,Z 335.596,A -85,B 0,C 180,E1 -5448.577,E2 -5448.577} C_VEL
LIN {X 0,Y 509.854,Z 335.598,A -85,B 0,C 180,E1 -5451.664,E2 -5451.664} C_VEL
LIN {X 0,Y 509.842,Z 335.599,A -85,B 0,C 180,E1 -5454.625,E2 -5454.625} C_VEL
LIN {X 0,Y 509.863,Z 335.596,A -85,B 0,C 180,E1 -5457.482,E2 -5457.482} C_VEL
LIN {X 0,Y 509.878,Z 335.584,A -85,B 0,C 180,E1 -5460.27,E2 -5460.27} C_VEL
LIN {X 0,Y 509.885,Z 335.597,A -85,B 0,C 180,E1 -5462.946,E2 -5462.946} C_VEL
LIN {X 0,Y 509.92,Z 335.739,A -85,B 0,C 180,E1 -5465.111,E2 -5465.111} C_VEL
LIN {X 0,Y 511.887,Z 345.824,A -85,B 0,C 180,E1 -5466.909,E2 -5466.909} C_VEL
LIN {X 0,Y 511.38,Z 362.105,A -85,B 0,C 180,E1 -5469.525,E2 -5469.525} C_VEL
LIN {X 0,Y 511.065,Z 372.2,A -85,B 0,C 180,E1 -5471.094,E2 -5471.094} C_VEL
LIN {X 0,Y 513.638,Z 385.912,A -85,B 0,C 180,E1 -5471.418,E2 -5471.418} C_VEL
LIN {X 0,Y 512.885,Z 508.696,A -85,B 0,C 180,E1 -5473.175,E2 -5473.175} C_VEL
LIN {X 0,Y 512.613,Z 522.978,A -85,B 0,C 180,E1 -5473.528,E2 -5473.528} C_VEL
LIN {X 0,Y 512.379,Z 535.838,A -85,B 0,C 180,E1 -5473.994,E2 -5473.994} C_VEL
LIN {X 0,Y 511.962,Z 548.116,A -85,B 0,C 180,E1 -5474.576,E2 -5474.576} C_VEL
LIN {X 0,Y 511.492,Z 561.265,A -85,B 0,C 180,E1 -5475.377,E2 -5475.377} C_VEL
LIN {X 0,Y 511.031,Z 573.144,A -85,B 0,C 180,E1 -5476.278,E2 -5476.278} C_VEL
LIN {X 0,Y 510.541,Z 585.025,A -85,B 0,C 180,E1 -5477.384,E2 -5477.384} C_VEL
LIN {X 0,Y 510.263,Z 594.715,A -85,B 0,C 180,E1 -5478.481,E2 -5478.481} C_VEL
LIN {X 0,Y 509.851,Z 603.563,A -85,B 0,C 180,E1 -5479.678,E2 -5479.678} C_VEL
LIN {X 0,Y 509.623,Z 610.925,A -85,B 0,C 180,E1 -5480.876,E2 -5480.876} C_VEL
LIN {X 0,Y 509.449,Z 617.058,A -85,B 0,C 180,E1 -5482.072,E2 -5482.072} C_VEL
LIN {X 0,Y 509.311,Z 623.571,A -85,B 0,C 180,E1 -5483.663,E2 -5483.663} C_VEL
LIN {X 0,Y 509.238,Z 627.384,A -85,B 0,C 180,E1 -5484.854,E2 -5484.854} C_VEL
LIN {X 0,Y 509.219,Z 630.322,A -85,B 0,C 180,E1 -5486.044,E2 -5486.044} C_VEL
LIN {X 0,Y 509.159,Z 633.007,A -85,B 0,C 180,E1 -5487.628,E2 -5487.628} C_VEL
LIN {X 0,Y 509.071,Z 634.335,A -85,B 0,C 180,E1 -5489.21,E2 -5489.21} C_VEL
LIN {X 0,Y 509.071,Z 634.333,A -85,B 0,C 180,E1 -5490.792,E2 -5490.792} C_VEL
LIN {X 0,Y 509.159,Z 633.001,A -85,B 0,C 180,E1 -5492.374,E2 -5492.374} C_VEL
LIN {X 0,Y 509.219,Z 630.313,A -85,B 0,C 180,E1 -5493.958,E2 -5493.958} C_VEL
LIN {X 0,Y 509.301,Z 626.197,A -85,B 0,C 180,E1 -5495.544,E2 -5495.544} C_VEL
LIN {X 0,Y 509.331,Z 620.524,A -85,B 0,C 180,E1 -5497.135,E2 -5497.135} C_VEL
LIN {X 0,Y 509.554,Z 614.121,A -85,B 0,C 180,E1 -5498.528,E2 -5498.528} C_VEL
LIN {X 0,Y 509.788,Z 606.168,A -85,B 0,C 180,E1 -5499.924,E2 -5499.924} C_VEL
LIN {X 0,Y 510.115,Z 597.845,A -85,B 0,C 180,E1 -5501.122,E2 -5501.122} C_VEL
LIN {X 0,Y 510.466,Z 587.749,A -85,B 0,C 180,E1 -5502.331,E2 -5502.331} C_VEL
LIN {X 0,Y 510.908,Z 576.64,A -85,B 0,C 180,E1 -5503.423,E2 -5503.423} C_VEL
LIN {X 0,Y 511.351,Z 564.083,A -85,B 0,C 180,E1 -5504.426,E2 -5504.426} C_VEL
LIN {X 0,Y 511.859,Z 551.62,A -85,B 0,C 180,E1 -5505.225,E2 -5505.225} C_VEL
LIN {X 0,Y 512.221,Z 538.813,A -85,B 0,C 180,E1 -5505.877,E2 -5505.877} C_VEL
LIN {X 0,Y 512.573,Z 524.674,A -85,B 0,C 180,E1 -5506.417,E2 -5506.417} C_VEL
LIN {X 0,Y 512.853,Z 510.985,A -85,B 0,C 180,E1 -5506.777,E2 -5506.777} C_VEL
LIN {X 0,Y 513.104,Z 482.876,A -85,B 0,C 180,E1 -5507.205,E2 -5507.205} C_VEL
LIN {X 0,Y 513.631,Z 385.888,A -85,B 0,C 180,E1 -5508.582,E2 -5508.582} C_VEL
LIN {X 0,Y 511.073,Z 372.187,A -85,B 0,C 180,E1 -5508.906,E2 -5508.906} C_VEL
LIN {X 0,Y 511.651,Z 354.006,A -85,B 0,C 180,E1 -5511.77,E2 -5511.77} C_VEL
LIN {X 0,Y 511.817,Z 345.094,A -85,B 0,C 180,E1 -5513.214,E2 -5513.214} C_VEL
LIN {X 0,Y 509.927,Z 335.723,A -85,B 0,C 180,E1 -5514.892,E2 -5514.892} C_VEL
LIN {X 0,Y 509.899,Z 335.59,A -85,B 0,C 180,E1 -5517.946,E2 -5517.946} C_VEL
LIN {X 0,Y 509.85,Z 335.6,A -85,B 0,C 180,E1 -5520.666,E2 -5520.666} C_VEL
LIN {X 0,Y 509.866,Z 335.597,A -85,B 0,C 180,E1 -5523.461,E2 -5523.461} C_VEL
LIN {X 0,Y 509.841,Z 335.604,A -85,B 0,C 180,E1 -5526.353,E2 -5526.353} C_VEL
LIN {X 0,Y 509.838,Z 335.602,A -85,B 0,C 180,E1 -5529.471,E2 -5529.471} C_VEL
LIN {X 0,Y 509.837,Z 335.6,A -85,B 0,C 180,E1 -5532.49,E2 -5532.49} C_VEL
LIN {X 0,Y 509.844,Z 335.6,A -85,B 0,C 180,E1 -5535.331,E2 -5535.331} C_VEL
LIN {X 0,Y 509.861,Z 335.598,A -85,B 0,C 180,E1 -5538.575,E2 -5538.575} C_VEL
LIN {X 0,Y 509.855,Z 335.604,A -85,B 0,C 180,E1 -5541.787,E2 -5541.787} C_VEL
LIN {X 0,Y 509.834,Z 335.6,A -85,B 0,C 180,E1 -5544.622,E2 -5544.622} C_VEL
LIN {X 0,Y 509.866,Z 335.602,A -85,B 0,C 180,E1 -5547.481,E2 -5547.481} C_VEL
LIN {X 0,Y 509.863,Z 335.6,A -85,B 0,C 180,E1 -5550.274,E2 -5550.274} C_VEL
LIN {X 0,Y 509.971,Z 335.815,A -85,B 0,C 180,E1 -5553.325,E2 -5553.325} C_VEL
LIN {X 0,Y 511.895,Z 346.556,A -85,B 0,C 180,E1 -5554.811,E2 -5554.811} C_VEL
LIN {X 0,Y 511.558,Z 369.787,A -85,B 0,C 180,E1 -5557.802,E2 -5557.802} C_VEL
LIN {X 0,Y 511.148,Z 390.73,A -85,B 0,C 180,E1 -5560.523,E2 -5560.523} C_VEL
LIN {X 0,Y 510.781,Z 412.835,A -85,B 0,C 180,E1 -5563.411,E2 -5563.411} C_VEL
LIN {X 0,Y 510.622,Z 421.038,A -85,B 0,C 180,E1 -5564.464,E2 -5564.464} C_VEL
LIN {X 0,Y 512.195,Z 433.036,A -85,B 0,C 180,E1 -5564.717,E2 -5564.717} C_VEL
LIN {X 0,Y 511.541,Z 530.839,A -85,B 0,C 180,E1 -5566.189,E2 -5566.189} C_VEL
LIN {X 0,Y 511.367,Z 543.262,A -85,B 0,C 180,E1 -5566.514,E2 -5566.514} C_VEL
LIN {X 0,Y 511.061,Z 555.529,A -85,B 0,C 180,E1 -5566.986,E2 -5566.986} C_VEL
LIN {X 0,Y 510.777,Z 568.451,A -85,B 0,C 180,E1 -5567.668,E2 -5567.668} C_VEL
LIN {X 0,Y 510.513,Z 579.016,A -85,B 0,C 180,E1 -5568.385,E2 -5568.385} C_VEL
LIN {X 0,Y 510.181,Z 589.584,A -85,B 0,C 180,E1 -5569.282,E2 -5569.282} C_VEL
LIN {X 0,Y 509.919,Z 599.115,A -85,B 0,C 180,E1 -5570.28,E2 -5570.28} C_VEL
LIN {X 0,Y 509.7,Z 606.933,A -85,B 0,C 180,E1 -5571.276,E2 -5571.276} C_VEL
LIN {X 0,Y 509.473,Z 614.571,A -85,B 0,C 180,E1 -5572.47,E2 -5572.47} C_VEL
LIN {X 0,Y 509.321,Z 620.674,A -85,B 0,C 180,E1 -5573.662,E2 -5573.662} C_VEL
LIN {X 0,Y 509.248,Z 625.503,A -85,B 0,C 180,E1 -5574.853,E2 -5574.853} C_VEL
LIN {X 0,Y 509.25,Z 629.198,A -85,B 0,C 180,E1 -5576.043,E2 -5576.043} C_VEL
LIN {X 0,Y 509.201,Z 631.099,A -85,B 0,C 180,E1 -5576.835,E2 -5576.835} C_VEL
LIN {X 0,Y 509.161,Z 632.563,A -85,B 0,C 180,E1 -5577.627,E2 -5577.627} C_VEL
LIN {X 0,Y 509.074,Z 634.212,A -85,B 0,C 180,E1 -5579.209,E2 -5579.209} C_VEL
LIN {X 0,Y 509.066,Z 634.457,A -85,B 0,C 180,E1 -5580,E2 -5580} C_VEL
LIN {X 0,Y 509.074,Z 634.268,A -85,B 0,C 180,E1 -5580.791,E2 -5580.791} C_VEL
LIN {X 0,Y 509.161,Z 632.695,A -85,B 0,C 180,E1 -5582.373,E2 -5582.373} C_VEL
LIN {X 0,Y 509.201,Z 631.306,A -85,B 0,C 180,E1 -5583.165,E2 -5583.165} C_VEL
LIN {X 0,Y 509.222,Z 628.389,A -85,B 0,C 180,E1 -5584.353,E2 -5584.353} C_VEL
LIN {X 0,Y 509.314,Z 624.421,A -85,B 0,C 180,E1 -5585.543,E2 -5585.543} C_VEL
LIN {X 0,Y 509.402,Z 618.739,A -85,B 0,C 180,E1 -5586.844,E2 -5586.844} C_VEL
LIN {X 0,Y 509.568,Z 611.602,A -85,B 0,C 180,E1 -5588.127,E2 -5588.127} C_VEL
LIN {X 0,Y 509.779,Z 603.239,A -85,B 0,C 180,E1 -5589.322,E2 -5589.322} C_VEL
LIN {X 0,Y 510.015,Z 594.645,A -85,B 0,C 180,E1 -5590.32,E2 -5590.32} C_VEL
LIN {X 0,Y 510.395,Z 584.117,A -85,B 0,C 180,E1 -5591.316,E2 -5591.316} C_VEL
LIN {X 0,Y 510.704,Z 573.588,A -85,B 0,C 180,E1 -5592.114,E2 -5592.114} C_VEL
LIN {X 0,Y 510.956,Z 561.935,A -85,B 0,C 180,E1 -5592.814,E2 -5592.814} C_VEL
LIN {X 0,Y 511.253,Z 550.019,A -85,B 0,C 180,E1 -5593.363,E2 -5593.363} C_VEL
LIN {X 0,Y 511.504,Z 536.994,A -85,B 0,C 180,E1 -5593.786,E2 -5593.786} C_VEL
LIN {X 0,Y 511.658,Z 523.245,A -85,B 0,C 180,E1 -5594.061,E2 -5594.061} C_VEL
LIN {X 0,Y 512.117,Z 431.086,A -85,B 0,C 180,E1 -5595.418,E2 -5595.418} C_VEL
LIN {X 0,Y 510.658,Z 421.038,A -85,B 0,C 180,E1 -5595.641,E2 -5595.641} C_VEL
LIN {X 0,Y 511.169,Z 396.909,A -85,B 0,C 180,E1 -5598.851,E2 -5598.851} C_VEL
LIN {X 0,Y 511.713,Z 373.649,A -85,B 0,C 180,E1 -5601.979,E2 -5601.979} C_VEL
LIN {X 0,Y 512.269,Z 353.285,A -85,B 0,C 180,E1 -5604.726,E2 -5604.726} C_VEL
LIN {X 0,Y 512.202,Z 346.836,A -85,B 0,C 180,E1 -5605.608,E2 -5605.608} C_VEL
LIN {X 0,Y 509.926,Z 335.704,A -85,B 0,C 180,E1 -5607.275,E2 -5607.275} C_VEL
LIN {X 0,Y 509.863,Z 335.6,A -85,B 0,C 180,E1 -5609.751,E2 -5609.751} C_VEL
LIN {X 0,Y 509.878,Z 335.598,A -85,B 0,C 180,E1 -5612.774,E2 -5612.774} C_VEL
LIN {X 0,Y 509.857,Z 335.603,A -85,B 0,C 180,E1 -5614.279,E2 -5614.279} C_VEL
LIN {X 0,Y 509.168,Z 335.69,A -85,B 0,C 180,E1 -5614.938,E2 -5614.938} C_VEL
LIN {X 0,Y 506.285,Z 336.045,A -85,B 0,C 180,E1 -5616.006,E2 -5616.006} C_VEL
LIN {X 0,Y 503.871,Z 336.344,A -85,B 0,C 180,E1 -5616.867,E2 -5616.867} C_VEL
LIN {X 0,Y 502.857,Z 336.469,A -85,B 0,C 180,E1 -5617.532,E2 -5617.532} C_VEL
LIN {X 0,Y 502.785,Z 336.479,A -85,B 0,C 180,E1 -5617.757,E2 -5617.757} C_VEL
LIN {X 0,Y 502.823,Z 336.473,A -85,B 0,C 180,E1 -5620.995,E2 -5620.995} C_VEL
LIN {X 0,Y 502.784,Z 336.472,A -85,B 0,C 180,E1 -5624.34,E2 -5624.34} C_VEL
LIN {X 0,Y 502.779,Z 336.479,A -85,B 0,C 180,E1 -5626.768,E2 -5626.768} C_VEL
LIN {X 0,Y 502.823,Z 336.47,A -85,B 0,C 180,E1 -5629.005,E2 -5629.005} C_VEL
LIN {X 0,Y 502.799,Z 336.482,A -85,B 0,C 180,E1 -5632.046,E2 -5632.046} C_VEL
LIN {X 0,Y 502.813,Z 336.473,A -85,B 0,C 180,E1 -5635.034,E2 -5635.034} C_VEL
LIN {X 0,Y 502.789,Z 336.48,A -85,B 0,C 180,E1 -5637.915,E2 -5637.915} C_VEL
LIN {X 0,Y 502.83,Z 336.458,A -85,B 0,C 180,E1 -5640.712,E2 -5640.712} C_VEL
LIN {X 0,Y 502.868,Z 336.467,A -85,B 0,C 180,E1 -5643.439,E2 -5643.439} C_VEL
LIN {X 0,Y 502.876,Z 336.659,A -85,B 0,C 180,E1 -5644.952,E2 -5644.952} C_VEL
LIN {X 0,Y 504.904,Z 346.539,A -85,B 0,C 180,E1 -5646.735,E2 -5646.735} C_VEL
LIN {X 0,Y 504.712,Z 356.345,A -85,B 0,C 180,E1 -5648.345,E2 -5648.345} C_VEL
LIN {X 0,Y 504.159,Z 372.263,A -85,B 0,C 180,E1 -5650.876,E2 -5650.876} C_VEL
LIN {X 0,Y 506.943,Z 387.473,A -85,B 0,C 180,E1 -5651.232,E2 -5651.232} C_VEL
LIN {X 0,Y 506.095,Z 508.961,A -85,B 0,C 180,E1 -5652.992,E2 -5652.992} C_VEL
LIN {X 0,Y 505.788,Z 523.714,A -85,B 0,C 180,E1 -5653.369,E2 -5653.369} C_VEL
LIN {X 0,Y 505.447,Z 537.833,A -85,B 0,C 180,E1 -5653.905,E2 -5653.905} C_VEL
LIN {X 0,Y 505.042,Z 550.852,A -85,B 0,C 180,E1 -5654.565,E2 -5654.565} C_VEL
LIN {X 0,Y 504.48,Z 563.461,A -85,B 0,C 180,E1 -5655.373,E2 -5655.373} C_VEL
LIN {X 0,Y 504.022,Z 574.954,A -85,B 0,C 180,E1 -5656.287,E2 -5656.287} C_VEL
LIN {X 0,Y 503.52,Z 585.693,A -85,B 0,C 180,E1 -5657.32,E2 -5657.32} C_VEL
LIN {X 0,Y 503.206,Z 595.967,A -85,B 0,C 180,E1 -5658.519,E2 -5658.519} C_VEL
LIN {X 0,Y 502.793,Z 604.604,A -85,B 0,C 180,E1 -5659.733,E2 -5659.733} C_VEL
LIN {X 0,Y 502.529,Z 612.885,A -85,B 0,C 180,E1 -5661.15,E2 -5661.15} C_VEL
LIN {X 0,Y 502.335,Z 618.657,A -85,B 0,C 180,E1 -5662.361,E2 -5662.361} C_VEL
LIN {X 0,Y 502.236,Z 623.407,A -85,B 0,C 180,E1 -5663.571,E2 -5663.571} C_VEL
LIN {X 0,Y 502.174,Z 627.258,A -85,B 0,C 180,E1 -5664.78,E2 -5664.78} C_VEL
LIN {X 0,Y 502.116,Z 630.213,A -85,B 0,C 180,E1 -5665.986,E2 -5665.986} C_VEL
LIN {X 0,Y 502.064,Z 632.938,A -85,B 0,C 180,E1 -5667.592,E2 -5667.592} C_VEL
LIN {X 0,Y 501.987,Z 634.309,A -85,B 0,C 180,E1 -5669.197,E2 -5669.197} C_VEL
LIN {X 0,Y 501.988,Z 634.353,A -85,B 0,C 180,E1 -5670.801,E2 -5670.801} C_VEL
LIN {X 0,Y 502.063,Z 633.068,A -85,B 0,C 180,E1 -5672.406,E2 -5672.406} C_VEL
LIN {X 0,Y 502.115,Z 630.422,A -85,B 0,C 180,E1 -5674.012,E2 -5674.012} C_VEL
LIN {X 0,Y 502.226,Z 626.343,A -85,B 0,C 180,E1 -5675.62,E2 -5675.62} C_VEL
LIN {X 0,Y 502.254,Z 620.71,A -85,B 0,C 180,E1 -5677.234,E2 -5677.234} C_VEL
LIN {X 0,Y 502.5,Z 614.356,A -85,B 0,C 180,E1 -5678.646,E2 -5678.646} C_VEL
LIN {X 0,Y 502.72,Z 606.453,A -85,B 0,C 180,E1 -5680.063,E2 -5680.063} C_VEL
LIN {X 0,Y 503.095,Z 598.187,A -85,B 0,C 180,E1 -5681.277,E2 -5681.277} C_VEL
LIN {X 0,Y 503.51,Z 587.608,A -85,B 0,C 180,E1 -5682.565,E2 -5682.565} C_VEL
LIN {X 0,Y 503.977,Z 576.004,A -85,B 0,C 180,E1 -5683.712,E2 -5683.712} C_VEL
LIN {X 0,Y 504.455,Z 564.737,A -85,B 0,C 180,E1 -5684.625,E2 -5684.625} C_VEL
LIN {X 0,Y 504.933,Z 552.426,A -85,B 0,C 180,E1 -5685.437,E2 -5685.437} C_VEL
LIN {X 0,Y 505.407,Z 539.829,A -85,B 0,C 180,E1 -5686.095,E2 -5686.095} C_VEL
LIN {X 0,Y 505.762,Z 525.443,A -85,B 0,C 180,E1 -5686.663,E2 -5686.663} C_VEL
LIN {X 0,Y 506.038,Z 511.905,A -85,B 0,C 180,E1 -5687.034,E2 -5687.034} C_VEL
LIN {X 0,Y 506.278,Z 489.688,A -85,B 0,C 180,E1 -5687.39,E2 -5687.39} C_VEL
LIN {X 0,Y 506.852,Z 386.298,A -85,B 0,C 180,E1 -5688.879,E2 -5688.879} C_VEL
LIN {X 0,Y 504.184,Z 372.391,A -85,B 0,C 180,E1 -5689.207,E2 -5689.207} C_VEL
LIN {X 0,Y 504.287,Z 367.373,A -85,B 0,C 180,E1 -5689.964,E2 -5689.964} C_VEL
LIN {X 0,Y 505.033,Z 347.774,A -85,B 0,C 180,E1 -5693.145,E2 -5693.145} C_VEL
LIN {X 0,Y 502.886,Z 336.591,A -85,B 0,C 180,E1 -5695.167,E2 -5695.167} C_VEL
LIN {X 0,Y 502.834,Z 336.476,A -85,B 0,C 180,E1 -5697.465,E2 -5697.465} C_VEL
LIN {X 0,Y 502.817,Z 336.469,A -85,B 0,C 180,E1 -5700.209,E2 -5700.209} C_VEL
LIN {X 0,Y 502.829,Z 336.47,A -85,B 0,C 180,E1 -5703.03,E2 -5703.03} C_VEL
LIN {X 0,Y 502.779,Z 336.479,A -85,B 0,C 180,E1 -5705.949,E2 -5705.949} C_VEL
LIN {X 0,Y 502.817,Z 336.471,A -85,B 0,C 180,E1 -5708.973,E2 -5708.973} C_VEL
LIN {X 0,Y 502.817,Z 336.478,A -85,B 0,C 180,E1 -5712.201,E2 -5712.201} C_VEL
LIN {X 0,Y 502.794,Z 336.469,A -85,B 0,C 180,E1 -5715.467,E2 -5715.467} C_VEL
LIN {X 0,Y 502.832,Z 336.478,A -85,B 0,C 180,E1 -5717.864,E2 -5717.864} C_VEL
LIN {X 0,Y 502.814,Z 336.468,A -85,B 0,C 180,E1 -5721.025,E2 -5721.025} C_VEL
LIN {X 0,Y 502.778,Z 336.478,A -85,B 0,C 180,E1 -5724.166,E2 -5724.166} C_VEL
LIN {X 0,Y 502.824,Z 336.473,A -85,B 0,C 180,E1 -5726.992,E2 -5726.992} C_VEL
LIN {X 0,Y 502.822,Z 336.457,A -85,B 0,C 180,E1 -5730.061,E2 -5730.061} C_VEL
LIN {X 0,Y 502.827,Z 336.461,A -85,B 0,C 180,E1 -5732.533,E2 -5732.533} C_VEL
LIN {X 0,Y 502.822,Z 336.476,A -85,B 0,C 180,E1 -5735.297,E2 -5735.297} C_VEL
LIN {X 0,Y 502.801,Z 336.473,A -85,B 0,C 180,E1 -5737.827,E2 -5737.827} C_VEL
LIN {X 0,Y 502.816,Z 336.471,A -85,B 0,C 180,E1 -5740.4,E2 -5740.4} C_VEL
LIN {X 0,Y 502.827,Z 336.473,A -85,B 0,C 180,E1 -5742.931,E2 -5742.931} C_VEL
LIN {X 0,Y 502.841,Z 336.473,A -85,B 0,C 180,E1 -5745.429,E2 -5745.429} C_VEL
LIN {X 0,Y 502.888,Z 336.464,A -85,B 0,C 180,E1 -5748.717,E2 -5748.717} C_VEL
LIN {X 0,Y 502.892,Z 336.461,A -85,B 0,C 180,E1 -5751.966,E2 -5751.966} C_VEL
LIN {X 0,Y 502.939,Z 336.457,A -85,B 0,C 180,E1 -5754.386,E2 -5754.386} C_VEL
LIN {X 0,Y 503.016,Z 336.447,A -85,B 0,C 180,E1 -5757.598,E2 -5757.598} C_VEL
LIN {X 0,Y 503.016,Z 336.448,A -85,B 0,C 180,E1 -5760,E2 -5760} C_VEL
LIN {X 0,Y 503.016,Z 336.447,A -85,B 0,C 180,E1 -5762.402,E2 -5762.402} C_VEL
LIN {X 0,Y 502.939,Z 336.457,A -85,B 0,C 180,E1 -5765.613,E2 -5765.613} C_VEL
LIN {X 0,Y 502.892,Z 336.461,A -85,B 0,C 180,E1 -5768.033,E2 -5768.033} C_VEL
LIN {X 0,Y 502.887,Z 336.464,A -85,B 0,C 180,E1 -5771.283,E2 -5771.283} C_VEL
LIN {X 0,Y 502.841,Z 336.473,A -85,B 0,C 180,E1 -5774.571,E2 -5774.571} C_VEL
LIN {X 0,Y 502.852,Z 336.467,A -85,B 0,C 180,E1 -5777.907,E2 -5777.907} C_VEL
LIN {X 0,Y 502.82,Z 336.475,A -85,B 0,C 180,E1 -5780.537,E2 -5780.537} C_VEL
LIN {X 0,Y 502.796,Z 336.478,A -85,B 0,C 180,E1 -5783.04,E2 -5783.04} C_VEL
LIN {X 0,Y 502.832,Z 336.469,A -85,B 0,C 180,E1 -5785.676,E2 -5785.676} C_VEL
LIN {X 0,Y 502.831,Z 336.459,A -85,B 0,C 180,E1 -5788.373,E2 -5788.373} C_VEL
LIN {X 0,Y 502.787,Z 336.472,A -85,B 0,C 180,E1 -5791.5,E2 -5791.5} C_VEL
LIN {X 0,Y 502.798,Z 336.48,A -85,B 0,C 180,E1 -5794.446,E2 -5794.446} C_VEL
LIN {X 0,Y 502.772,Z 336.466,A -85,B 0,C 180,E1 -5797.179,E2 -5797.179} C_VEL
LIN {X 0,Y 502.814,Z 336.472,A -85,B 0,C 180,E1 -5800.013,E2 -5800.013} C_VEL
LIN {X 0,Y 502.82,Z 336.479,A -85,B 0,C 180,E1 -5802.203,E2 -5802.203} C_VEL
LIN {X 0,Y 502.793,Z 336.468,A -85,B 0,C 180,E1 -5805.469,E2 -5805.469} C_VEL
LIN {X 0,Y 502.829,Z 336.477,A -85,B 0,C 180,E1 -5807.866,E2 -5807.866} C_VEL
LIN {X 0,Y 502.816,Z 336.471,A -85,B 0,C 180,E1 -5811.027,E2 -5811.027} C_VEL
LIN {X 0,Y 502.781,Z 336.479,A -85,B 0,C 180,E1 -5814.168,E2 -5814.168} C_VEL
LIN {X 0,Y 502.829,Z 336.47,A -85,B 0,C 180,E1 -5816.994,E2 -5816.994} C_VEL
LIN {X 0,Y 502.827,Z 336.464,A -85,B 0,C 180,E1 -5820.063,E2 -5820.063} C_VEL
LIN {X 0,Y 502.833,Z 336.476,A -85,B 0,C 180,E1 -5822.535,E2 -5822.535} C_VEL
LIN {X 0,Y 502.862,Z 336.632,A -85,B 0,C 180,E1 -5824.892,E2 -5824.892} C_VEL
LIN {X 0,Y 505.028,Z 347.587,A -85,B 0,C 180,E1 -5826.869,E2 -5826.869} C_VEL
LIN {X 0,Y 504.329,Z 365.788,A -85,B 0,C 180,E1 -5829.826,E2 -5829.826} C_VEL
LIN {X 0,Y 504.176,Z 372.195,A -85,B 0,C 180,E1 -5830.826,E2 -5830.826} C_VEL
LIN {X 0,Y 506.806,Z 386.207,A -85,B 0,C 180,E1 -5831.163,E2 -5831.163} C_VEL
LIN {X 0,Y 506.818,Z 414.375,A -85,B 0,C 180,E1 -5831.576,E2 -5831.576} C_VEL
LIN {X 0,Y 506.061,Z 509.934,A -85,B 0,C 180,E1 -5832.967,E2 -5832.967} C_VEL
LIN {X 0,Y 505.778,Z 524.136,A -85,B 0,C 180,E1 -5833.338,E2 -5833.338} C_VEL
LIN {X 0,Y 505.452,Z 537.719,A -85,B 0,C 180,E1 -5833.855,E2 -5833.855} C_VEL
LIN {X 0,Y 505.061,Z 549.89,A -85,B 0,C 180,E1 -5834.464,E2 -5834.464} C_VEL
LIN {X 0,Y 504.538,Z 562.69,A -85,B 0,C 180,E1 -5835.274,E2 -5835.274} C_VEL
LIN {X 0,Y 504.051,Z 574.318,A -85,B 0,C 180,E1 -5836.187,E2 -5836.187} C_VEL
LIN {X 0,Y 503.531,Z 585.948,A -85,B 0,C 180,E1 -5837.302,E2 -5837.302} C_VEL
LIN {X 0,Y 503.209,Z 596.342,A -85,B 0,C 180,E1 -5838.521,E2 -5838.521} C_VEL
LIN {X 0,Y 502.79,Z 604.916,A -85,B 0,C 180,E1 -5839.735,E2 -5839.735} C_VEL
LIN {X 0,Y 502.51,Z 613.125,A -85,B 0,C 180,E1 -5841.151,E2 -5841.151} C_VEL
LIN {X 0,Y 502.32,Z 618.866,A -85,B 0,C 180,E1 -5842.363,E2 -5842.363} C_VEL
LIN {X 0,Y 502.233,Z 623.571,A -85,B 0,C 180,E1 -5843.573,E2 -5843.573} C_VEL
LIN {X 0,Y 502.172,Z 627.384,A -85,B 0,C 180,E1 -5844.782,E2 -5844.782} C_VEL
LIN {X 0,Y 502.115,Z 630.322,A -85,B 0,C 180,E1 -5845.988,E2 -5845.988} C_VEL
LIN {X 0,Y 502.063,Z 633.007,A -85,B 0,C 180,E1 -5847.594,E2 -5847.594} C_VEL
LIN {X 0,Y 501.988,Z 634.335,A -85,B 0,C 180,E1 -5849.199,E2 -5849.199} C_VEL
LIN {X 0,Y 501.988,Z 634.333,A -85,B 0,C 180,E1 -5850.803,E2 -5850.803} C_VEL
LIN {X 0,Y 502.063,Z 633.001,A -85,B 0,C 180,E1 -5852.408,E2 -5852.408} C_VEL
LIN {X 0,Y 502.115,Z 630.313,A -85,B 0,C 180,E1 -5854.014,E2 -5854.014} C_VEL
LIN {X 0,Y 502.218,Z 626.197,A -85,B 0,C 180,E1 -5855.623,E2 -5855.623} C_VEL
LIN {X 0,Y 502.256,Z 620.524,A -85,B 0,C 180,E1 -5857.236,E2 -5857.236} C_VEL
LIN {X 0,Y 502.501,Z 614.121,A -85,B 0,C 180,E1 -5858.648,E2 -5858.648} C_VEL
LIN {X 0,Y 502.737,Z 606.168,A -85,B 0,C 180,E1 -5860.065,E2 -5860.065} C_VEL
LIN {X 0,Y 503.129,Z 597.845,A -85,B 0,C 180,E1 -5861.278,E2 -5861.278} C_VEL
LIN {X 0,Y 503.519,Z 587.187,A -85,B 0,C 180,E1 -5862.567,E2 -5862.567} C_VEL
LIN {X 0,Y 503.991,Z 576.64,A -85,B 0,C 180,E1 -5863.611,E2 -5863.611} C_VEL
LIN {X 0,Y 504.415,Z 565.508,A -85,B 0,C 180,E1 -5864.525,E2 -5864.525} C_VEL
LIN {X 0,Y 504.904,Z 553.385,A -85,B 0,C 180,E1 -5865.336,E2 -5865.336} C_VEL
LIN {X 0,Y 505.372,Z 539.943,A -85,B 0,C 180,E1 -5866.046,E2 -5866.046} C_VEL
LIN {X 0,Y 505.732,Z 525.914,A -85,B 0,C 180,E1 -5866.603,E2 -5866.603} C_VEL
LIN {X 0,Y 506.052,Z 512.125,A -85,B 0,C 180,E1 -5866.983,E2 -5866.983} C_VEL
LIN {X 0,Y 506.238,Z 491.819,A -85,B 0,C 180,E1 -5867.315,E2 -5867.315} C_VEL
LIN {X 0,Y 506.945,Z 387.004,A -85,B 0,C 180,E1 -5868.82,E2 -5868.82} C_VEL
LIN {X 0,Y 504.175,Z 372.306,A -85,B 0,C 180,E1 -5869.166,E2 -5869.166} C_VEL
LIN {X 0,Y 504.752,Z 355.313,A -85,B 0,C 180,E1 -5871.868,E2 -5871.868} C_VEL
LIN {X 0,Y 504.938,Z 346.746,A -85,B 0,C 180,E1 -5873.274,E2 -5873.274} C_VEL
LIN {X 0,Y 502.868,Z 336.614,A -85,B 0,C 180,E1 -5875.11,E2 -5875.11} C_VEL
LIN {X 0,Y 502.839,Z 336.475,A -85,B 0,C 180,E1 -5877.467,E2 -5877.467} C_VEL
LIN {X 0,Y 502.814,Z 336.477,A -85,B 0,C 180,E1 -5880.212,E2 -5880.212} C_VEL
LIN {X 0,Y 502.836,Z 336.471,A -85,B 0,C 180,E1 -5883.032,E2 -5883.032} C_VEL
LIN {X 0,Y 502.788,Z 336.483,A -85,B 0,C 180,E1 -5885.951,E2 -5885.951} C_VEL
LIN {X 0,Y 502.806,Z 336.476,A -85,B 0,C 180,E1 -5888.977,E2 -5888.977} C_VEL
LIN {X 0,Y 502.799,Z 336.48,A -85,B 0,C 180,E1 -5892.14,E2 -5892.14} C_VEL
LIN {X 0,Y 502.791,Z 336.48,A -85,B 0,C 180,E1 -5895.47,E2 -5895.47} C_VEL
LIN {X 0,Y 502.825,Z 336.474,A -85,B 0,C 180,E1 -5898.935,E2 -5898.935} C_VEL
LIN {X 0,Y 502.797,Z 336.481,A -85,B 0,C 180,E1 -5902.046,E2 -5902.046} C_VEL
LIN {X 0,Y 502.803,Z 336.478,A -85,B 0,C 180,E1 -5905.035,E2 -5905.035} C_VEL
LIN {X 0,Y 502.788,Z 336.484,A -85,B 0,C 180,E1 -5907.916,E2 -5907.916} C_VEL
LIN {X 0,Y 502.829,Z 336.476,A -85,B 0,C 180,E1 -5910.713,E2 -5910.713} C_VEL
LIN {X 0,Y 502.9,Z 336.676,A -85,B 0,C 180,E1 -5913.111,E2 -5913.111} C_VEL
LIN {X 0,Y 505.007,Z 347.769,A -85,B 0,C 180,E1 -5914.669,E2 -5914.669} C_VEL
LIN {X 0,Y 504.66,Z 369.384,A -85,B 0,C 180,E1 -5917.482,E2 -5917.482} C_VEL
LIN {X 0,Y 504.269,Z 388.82,A -85,B 0,C 180,E1 -5920.034,E2 -5920.034} C_VEL
LIN {X 0,Y 503.892,Z 409.589,A -85,B 0,C 180,E1 -5922.76,E2 -5922.76} C_VEL
LIN {X 0,Y 503.705,Z 421.174,A -85,B 0,C 180,E1 -5924.255,E2 -5924.255} C_VEL
LIN {X 0,Y 505.324,Z 433.2,A -85,B 0,C 180,E1 -5924.514,E2 -5924.514} C_VEL
LIN {X 0,Y 504.593,Z 532.017,A -85,B 0,C 180,E1 -5926.047,E2 -5926.047} C_VEL
LIN {X 0,Y 504.363,Z 544.713,A -85,B 0,C 180,E1 -5926.4,E2 -5926.4} C_VEL
LIN {X 0,Y 504.094,Z 557.07,A -85,B 0,C 180,E1 -5926.906,E2 -5926.906} C_VEL
LIN {X 0,Y 503.792,Z 569.071,A -85,B 0,C 180,E1 -5927.56,E2 -5927.56} C_VEL
LIN {X 0,Y 503.498,Z 579.945,A -85,B 0,C 180,E1 -5928.323,E2 -5928.323} C_VEL
LIN {X 0,Y 503.139,Z 590.355,A -85,B 0,C 180,E1 -5929.232,E2 -5929.232} C_VEL
LIN {X 0,Y 502.873,Z 598.898,A -85,B 0,C 180,E1 -5930.142,E2 -5930.142} C_VEL
LIN {X 0,Y 502.628,Z 606.763,A -85,B 0,C 180,E1 -5931.152,E2 -5931.152} C_VEL
LIN {X 0,Y 502.406,Z 614.456,A -85,B 0,C 180,E1 -5932.363,E2 -5932.363} C_VEL
LIN {X 0,Y 502.238,Z 620.591,A -85,B 0,C 180,E1 -5933.572,E2 -5933.572} C_VEL
LIN {X 0,Y 502.182,Z 625.445,A -85,B 0,C 180,E1 -5934.781,E2 -5934.781} C_VEL
LIN {X 0,Y 502.147,Z 629.159,A -85,B 0,C 180,E1 -5935.987,E2 -5935.987} C_VEL
LIN {X 0,Y 502.121,Z 631.068,A -85,B 0,C 180,E1 -5936.791,E2 -5936.791} C_VEL
LIN {X 0,Y 502.066,Z 632.54,A -85,B 0,C 180,E1 -5937.593,E2 -5937.593} C_VEL
LIN {X 0,Y 502.036,Z 633.564,A -85,B 0,C 180,E1 -5938.396,E2 -5938.396} C_VEL
LIN {X 0,Y 501.981,Z 634.444,A -85,B 0,C 180,E1 -5940,E2 -5940} C_VEL
LIN {X 0,Y 501.991,Z 634.253,A -85,B 0,C 180,E1 -5940.802,E2 -5940.802} C_VEL
LIN {X 0,Y 502.036,Z 633.657,A -85,B 0,C 180,E1 -5941.604,E2 -5941.604} C_VEL
LIN {X 0,Y 502.066,Z 632.671,A -85,B 0,C 180,E1 -5942.407,E2 -5942.407} C_VEL
LIN {X 0,Y 502.122,Z 631.274,A -85,B 0,C 180,E1 -5943.21,E2 -5943.21} C_VEL
LIN {X 0,Y 502.118,Z 628.342,A -85,B 0,C 180,E1 -5944.415,E2 -5944.415} C_VEL
LIN {X 0,Y 502.231,Z 624.354,A -85,B 0,C 180,E1 -5945.621,E2 -5945.621} C_VEL
LIN {X 0,Y 502.333,Z 618.297,A -85,B 0,C 180,E1 -5947.012,E2 -5947.012} C_VEL
LIN {X 0,Y 502.5,Z 611.48,A -85,B 0,C 180,E1 -5948.242,E2 -5948.242} C_VEL
LIN {X 0,Y 502.739,Z 603.072,A -85,B 0,C 180,E1 -5949.454,E2 -5949.454} C_VEL
LIN {X 0,Y 502.978,Z 594.437,A -85,B 0,C 180,E1 -5950.466,E2 -5950.466} C_VEL
LIN {X 0,Y 503.421,Z 583.863,A -85,B 0,C 180,E1 -5951.475,E2 -5951.475} C_VEL
LIN {X 0,Y 503.696,Z 573.253,A -85,B 0,C 180,E1 -5952.285,E2 -5952.285} C_VEL
LIN {X 0,Y 504.013,Z 561.524,A -85,B 0,C 180,E1 -5952.994,E2 -5952.994} C_VEL
LIN {X 0,Y 504.333,Z 549.492,A -85,B 0,C 180,E1 -5953.55,E2 -5953.55} C_VEL
LIN {X 0,Y 504.589,Z 536.185,A -85,B 0,C 180,E1 -5953.979,E2 -5953.979} C_VEL
LIN {X 0,Y 504.752,Z 521.893,A -85,B 0,C 180,E1 -5954.257,E2 -5954.257} C_VEL
LIN {X 0,Y 505.306,Z 432.187,A -85,B 0,C 180,E1 -5955.61,E2 -5955.61} C_VEL
LIN {X 0,Y 503.683,Z 421.041,A -85,B 0,C 180,E1 -5955.856,E2 -5955.856} C_VEL
LIN {X 0,Y 504.227,Z 398.295,A -85,B 0,C 180,E1 -5958.909,E2 -5958.909} C_VEL
LIN {X 0,Y 504.798,Z 374.91,A -85,B 0,C 180,E1 -5962.08,E2 -5962.08} C_VEL
LIN {X 0,Y 505.381,Z 354.674,A -85,B 0,C 180,E1 -5964.834,E2 -5964.834} C_VEL
LIN {X 0,Y 505.247,Z 347.944,A -85,B 0,C 180,E1 -5965.766,E2 -5965.766} C_VEL
LIN {X 0,Y 502.897,Z 336.602,A -85,B 0,C 180,E1 -5967.477,E2 -5967.477} C_VEL
LIN {X 0,Y 502.815,Z 336.48,A -85,B 0,C 180,E1 -5970.211,E2 -5970.211} C_VEL
LIN {X 0,Y 502.837,Z 336.473,A -85,B 0,C 180,E1 -5973.031,E2 -5973.031} C_VEL
LIN {X 0,Y 502.778,Z 336.481,A -85,B 0,C 180,E1 -5975.951,E2 -5975.951} C_VEL
LIN {X 0,Y 502.785,Z 336.479,A -85,B 0,C 180,E1 -5977.757,E2 -5977.757} C_VEL
LIN {X 0,Y 502.151,Z 336.563,A -85,B 0,C 180,E1 -5978.427,E2 -5978.427} C_VEL
LIN {X 0,Y 499.317,Z 336.914,A -85,B 0,C 180,E1 -5979.513,E2 -5979.513} C_VEL
LIN {X 0,Y 496.896,Z 337.217,A -85,B 0,C 180,E1 -5980.389,E2 -5980.389} C_VEL
LIN {X 0,Y 495.849,Z 337.342,A -85,B 0,C 180,E1 -5981.065,E2 -5981.065} C_VEL
LIN {X 0,Y 495.76,Z 337.352,A -85,B 0,C 180,E1 -5981.294,E2 -5981.294} C_VEL
LIN {X 0,Y 495.733,Z 337.354,A -85,B 0,C 180,E1 -5984.001,E2 -5984.001} C_VEL
LIN {X 0,Y 495.731,Z 337.356,A -85,B 0,C 180,E1 -5987.117,E2 -5987.117} C_VEL
LIN {X 0,Y 495.764,Z 337.351,A -85,B 0,C 180,E1 -5989.953,E2 -5989.953} C_VEL
LIN {X 0,Y 495.735,Z 337.357,A -85,B 0,C 180,E1 -5992.552,E2 -5992.552} C_VEL
LIN {X 0,Y 495.789,Z 337.35,A -85,B 0,C 180,E1 -5995.457,E2 -5995.457} C_VEL
LIN {X 0,Y 495.761,Z 337.357,A -85,B 0,C 180,E1 -5998.363,E2 -5998.363} C_VEL
LIN {X 0,Y 495.793,Z 337.337,A -85,B 0,C 180,E1 -6001.506,E2 -6001.506} C_VEL
LIN {X 0,Y 495.828,Z 337.353,A -85,B 0,C 180,E1 -6004.609,E2 -6004.609} C_VEL
LIN {X 0,Y 495.935,Z 338.047,A -85,B 0,C 180,E1 -6004.84,E2 -6004.84} C_VEL
LIN {X 0,Y 498.037,Z 348.505,A -85,B 0,C 180,E1 -6006.726,E2 -6006.726} C_VEL
LIN {X 0,Y 497.629,Z 361.634,A -85,B 0,C 180,E1 -6008.9,E2 -6008.9} C_VEL
LIN {X 0,Y 497.273,Z 372.332,A -85,B 0,C 180,E1 -6010.605,E2 -6010.605} C_VEL
LIN {X 0,Y 500.243,Z 389.036,A -85,B 0,C 180,E1 -6010.994,E2 -6010.994} C_VEL
LIN {X 0,Y 499.335,Z 508.994,A -85,B 0,C 180,E1 -6012.755,E2 -6012.755} C_VEL
LIN {X 0,Y 499.015,Z 523.535,A -85,B 0,C 180,E1 -6013.129,E2 -6013.129} C_VEL
LIN {X 0,Y 498.668,Z 536.718,A -85,B 0,C 180,E1 -6013.627,E2 -6013.627} C_VEL
LIN {X 0,Y 498.235,Z 549.099,A -85,B 0,C 180,E1 -6014.243,E2 -6014.243} C_VEL
LIN {X 0,Y 497.697,Z 562.045,A -85,B 0,C 180,E1 -6015.065,E2 -6015.065} C_VEL
LIN {X 0,Y 497.166,Z 573.788,A -85,B 0,C 180,E1 -6015.99,E2 -6015.99} C_VEL
LIN {X 0,Y 496.628,Z 584.627,A -85,B 0,C 180,E1 -6017.027,E2 -6017.027} C_VEL
LIN {X 0,Y 496.262,Z 594.621,A -85,B 0,C 180,E1 -6018.184,E2 -6018.184} C_VEL
LIN {X 0,Y 495.835,Z 603.254,A -85,B 0,C 180,E1 -6019.381,E2 -6019.381} C_VEL
LIN {X 0,Y 495.536,Z 611.784,A -85,B 0,C 180,E1 -6020.818,E2 -6020.818} C_VEL
LIN {X 0,Y 495.277,Z 618.66,A -85,B 0,C 180,E1 -6022.252,E2 -6022.252} C_VEL
LIN {X 0,Y 495.133,Z 624.37,A -85,B 0,C 180,E1 -6023.755,E2 -6023.755} C_VEL
LIN {X 0,Y 495.032,Z 628.323,A -85,B 0,C 180,E1 -6025.113,E2 -6025.113} C_VEL
LIN {X 0,Y 495.034,Z 631.749,A -85,B 0,C 180,E1 -6026.744,E2 -6026.744} C_VEL
LIN {X 0,Y 494.96,Z 633.79,A -85,B 0,C 180,E1 -6028.372,E2 -6028.372} C_VEL
LIN {X 0,Y 494.897,Z 634.497,A -85,B 0,C 180,E1 -6029.999,E2 -6029.999} C_VEL
LIN {X 0,Y 494.958,Z 633.877,A -85,B 0,C 180,E1 -6031.626,E2 -6031.626} C_VEL
LIN {X 0,Y 495.033,Z 631.917,A -85,B 0,C 180,E1 -6033.254,E2 -6033.254} C_VEL
LIN {X 0,Y 495.031,Z 628.567,A -85,B 0,C 180,E1 -6034.885,E2 -6034.885} C_VEL
LIN {X 0,Y 495.13,Z 624.688,A -85,B 0,C 180,E1 -6036.242,E2 -6036.242} C_VEL
LIN {X 0,Y 495.263,Z 619.065,A -85,B 0,C 180,E1 -6037.746,E2 -6037.746} C_VEL
LIN {X 0,Y 495.506,Z 612.284,A -85,B 0,C 180,E1 -6039.18,E2 -6039.18} C_VEL
LIN {X 0,Y 495.814,Z 603.858,A -85,B 0,C 180,E1 -6040.617,E2 -6040.617} C_VEL
LIN {X 0,Y 496.261,Z 594.143,A -85,B 0,C 180,E1 -6041.967,E2 -6041.967} C_VEL
LIN {X 0,Y 496.674,Z 584.417,A -85,B 0,C 180,E1 -6043.084,E2 -6043.084} C_VEL
LIN {X 0,Y 497.167,Z 573.65,A -85,B 0,C 180,E1 -6044.113,E2 -6044.113} C_VEL
LIN {X 0,Y 497.695,Z 561.877,A -85,B 0,C 180,E1 -6045.038,E2 -6045.038} C_VEL
LIN {X 0,Y 498.173,Z 548.88,A -85,B 0,C 180,E1 -6045.862,E2 -6045.862} C_VEL
LIN {X 0,Y 498.716,Z 535.514,A -85,B 0,C 180,E1 -6046.516,E2 -6046.516} C_VEL
LIN {X 0,Y 499.059,Z 521.433,A -85,B 0,C 180,E1 -6047.026,E2 -6047.026} C_VEL
LIN {X 0,Y 499.358,Z 506.752,A -85,B 0,C 180,E1 -6047.374,E2 -6047.374} C_VEL
LIN {X 0,Y 500.226,Z 387.704,A -85,B 0,C 180,E1 -6049.117,E2 -6049.117} C_VEL
LIN {X 0,Y 497.247,Z 372.214,A -85,B 0,C 180,E1 -6049.496,E2 -6049.496} C_VEL
LIN {X 0,Y 497.932,Z 354.291,A -85,B 0,C 180,E1 -6052.4,E2 -6052.4} C_VEL
LIN {X 0,Y 497.99,Z 347.95,A -85,B 0,C 180,E1 -6053.461,E2 -6053.461} C_VEL
LIN {X 0,Y 495.837,Z 337.494,A -85,B 0,C 180,E1 -6055.388,E2 -6055.388} C_VEL
LIN {X 0,Y 495.781,Z 337.351,A -85,B 0,C 180,E1 -6057.89,E2 -6057.89} C_VEL
LIN {X 0,Y 495.755,Z 337.357,A -85,B 0,C 180,E1 -6060.686,E2 -6060.686} C_VEL
LIN {X 0,Y 495.758,Z 337.352,A -85,B 0,C 180,E1 -6063.563,E2 -6063.563} C_VEL
LIN {X 0,Y 495.73,Z 337.358,A -85,B 0,C 180,E1 -6066.542,E2 -6066.542} C_VEL
LIN {X 0,Y 495.786,Z 337.348,A -85,B 0,C 180,E1 -6069.633,E2 -6069.633} C_VEL
LIN {X 0,Y 495.757,Z 337.353,A -85,B 0,C 180,E1 -6072.878,E2 -6072.878} C_VEL
LIN {X 0,Y 495.731,Z 337.353,A -85,B 0,C 180,E1 -6075.998,E2 -6075.998} C_VEL
LIN {X 0,Y 495.765,Z 337.352,A -85,B 0,C 180,E1 -6078.704,E2 -6078.704} C_VEL
LIN {X 0,Y 495.756,Z 337.347,A -85,B 0,C 180,E1 -6081.409,E2 -6081.409} C_VEL
LIN {X 0,Y 495.75,Z 337.351,A -85,B 0,C 180,E1 -6084.462,E2 -6084.462} C_VEL
LIN {X 0,Y 495.761,Z 337.357,A -85,B 0,C 180,E1 -6087.405,E2 -6087.405} C_VEL
LIN {X 0,Y 495.773,Z 337.333,A -85,B 0,C 180,E1 -6090.254,E2 -6090.254} C_VEL
LIN {X 0,Y 495.824,Z 337.337,A -85,B 0,C 180,E1 -6093.247,E2 -6093.247} C_VEL
LIN {X 0,Y 495.75,Z 337.358,A -85,B 0,C 180,E1 -6095.725,E2 -6095.725} C_VEL
LIN {X 0,Y 495.751,Z 337.348,A -85,B 0,C 180,E1 -6098.371,E2 -6098.371} C_VEL
LIN {X 0,Y 495.775,Z 337.351,A -85,B 0,C 180,E1 -6100.971,E2 -6100.971} C_VEL
LIN {X 0,Y 495.771,Z 337.349,A -85,B 0,C 180,E1 -6103.53,E2 -6103.53} C_VEL
LIN {X 0,Y 495.789,Z 337.346,A -85,B 0,C 180,E1 -6106.055,E2 -6106.055} C_VEL
LIN {X 0,Y 495.861,Z 337.338,A -85,B 0,C 180,E1 -6108.555,E2 -6108.555} C_VEL
LIN {X 0,Y 495.863,Z 337.337,A -85,B 0,C 180,E1 -6111.852,E2 -6111.852} C_VEL
LIN {X 0,Y 495.895,Z 337.334,A -85,B 0,C 180,E1 -6114.306,E2 -6114.306} C_VEL
LIN {X 0,Y 495.985,Z 337.323,A -85,B 0,C 180,E1 -6117.564,E2 -6117.564} C_VEL
LIN {X 0,Y 495.987,Z 337.323,A -85,B 0,C 180,E1 -6120,E2 -6120} C_VEL
LIN {X 0,Y 495.985,Z 337.323,A -85,B 0,C 180,E1 -6122.436,E2 -6122.436} C_VEL
LIN {X 0,Y 495.895,Z 337.335,A -85,B 0,C 180,E1 -6125.693,E2 -6125.693} C_VEL
LIN {X 0,Y 495.863,Z 337.337,A -85,B 0,C 180,E1 -6128.148,E2 -6128.148} C_VEL
LIN {X 0,Y 495.861,Z 337.338,A -85,B 0,C 180,E1 -6131.445,E2 -6131.445} C_VEL
LIN {X 0,Y 495.784,Z 337.348,A -85,B 0,C 180,E1 -6134.783,E2 -6134.783} C_VEL
LIN {X 0,Y 495.778,Z 337.349,A -85,B 0,C 180,E1 -6137.319,E2 -6137.319} C_VEL
LIN {X 0,Y 495.768,Z 337.349,A -85,B 0,C 180,E1 -6139.89,E2 -6139.89} C_VEL
LIN {X 0,Y 495.755,Z 337.357,A -85,B 0,C 180,E1 -6142.863,E2 -6142.863} C_VEL
LIN {X 0,Y 495.79,Z 337.348,A -85,B 0,C 180,E1 -6146.068,E2 -6146.068} C_VEL
LIN {X 0,Y 495.762,Z 337.334,A -85,B 0,C 180,E1 -6148.815,E2 -6148.815} C_VEL
LIN {X 0,Y 495.749,Z 337.349,A -85,B 0,C 180,E1 -6151.727,E2 -6151.727} C_VEL
LIN {X 0,Y 495.768,Z 337.352,A -85,B 0,C 180,E1 -6154.696,E2 -6154.696} C_VEL
LIN {X 0,Y 495.723,Z 337.344,A -85,B 0,C 180,E1 -6157.562,E2 -6157.562} C_VEL
LIN {X 0,Y 495.773,Z 337.353,A -85,B 0,C 180,E1 -6160.699,E2 -6160.699} C_VEL
LIN {X 0,Y 495.728,Z 337.355,A -85,B 0,C 180,E1 -6163.697,E2 -6163.697} C_VEL
LIN {X 0,Y 495.728,Z 337.359,A -85,B 0,C 180,E1 -6166.306,E2 -6166.306} C_VEL
LIN {X 0,Y 495.775,Z 337.348,A -85,B 0,C 180,E1 -6169.303,E2 -6169.303} C_VEL
LIN {X 0,Y 495.758,Z 337.352,A -85,B 0,C 180,E1 -6171.411,E2 -6171.411} C_VEL
LIN {X 0,Y 495.753,Z 337.355,A -85,B 0,C 180,E1 -6174.464,E2 -6174.464} C_VEL
LIN {X 0,Y 495.766,Z 337.351,A -85,B 0,C 180,E1 -6177.407,E2 -6177.407} C_VEL
LIN {X 0,Y 495.778,Z 337.339,A -85,B 0,C 180,E1 -6180.256,E2 -6180.256} C_VEL
LIN {X 0,Y 495.831,Z 337.345,A -85,B 0,C 180,E1 -6183.249,E2 -6183.249} C_VEL
LIN {X 0,Y 495.817,Z 337.388,A -85,B 0,C 180,E1 -6184.611,E2 -6184.611} C_VEL
LIN {X 0,Y 496.195,Z 339.311,A -85,B 0,C 180,E1 -6185.024,E2 -6185.024} C_VEL
LIN {X 0,Y 498.102,Z 348.792,A -85,B 0,C 180,E1 -6186.731,E2 -6186.731} C_VEL
LIN {X 0,Y 497.468,Z 365.789,A -85,B 0,C 180,E1 -6189.535,E2 -6189.535} C_VEL
LIN {X 0,Y 497.235,Z 372.194,A -85,B 0,C 180,E1 -6190.548,E2 -6190.548} C_VEL
LIN {X 0,Y 499.354,Z 383.226,A -85,B 0,C 180,E1 -6190.826,E2 -6190.826} C_VEL
LIN {X 0,Y 500.288,Z 388.997,A -85,B 0,C 180,E1 -6190.949,E2 -6190.949} C_VEL
LIN {X 0,Y 499.297,Z 509.934,A -85,B 0,C 180,E1 -6192.729,E2 -6192.729} C_VEL
LIN {X 0,Y 498.964,Z 524.514,A -85,B 0,C 180,E1 -6193.117,E2 -6193.117} C_VEL
LIN {X 0,Y 498.599,Z 538.848,A -85,B 0,C 180,E1 -6193.68,E2 -6193.68} C_VEL
LIN {X 0,Y 498.151,Z 551.657,A -85,B 0,C 180,E1 -6194.348,E2 -6194.348} C_VEL
LIN {X 0,Y 497.587,Z 564.115,A -85,B 0,C 180,E1 -6195.168,E2 -6195.168} C_VEL
LIN {X 0,Y 497.063,Z 575.491,A -85,B 0,C 180,E1 -6196.093,E2 -6196.093} C_VEL
LIN {X 0,Y 496.56,Z 585.948,A -85,B 0,C 180,E1 -6197.121,E2 -6197.121} C_VEL
LIN {X 0,Y 496.22,Z 596.442,A -85,B 0,C 180,E1 -6198.37,E2 -6198.37} C_VEL
LIN {X 0,Y 495.78,Z 604.916,A -85,B 0,C 180,E1 -6199.588,E2 -6199.588} C_VEL
LIN {X 0,Y 495.477,Z 613.125,A -85,B 0,C 180,E1 -6201.025,E2 -6201.025} C_VEL
LIN {X 0,Y 495.262,Z 618.866,A -85,B 0,C 180,E1 -6202.254,E2 -6202.254} C_VEL
LIN {X 0,Y 495.134,Z 624.517,A -85,B 0,C 180,E1 -6203.753,E2 -6203.753} C_VEL
LIN {X 0,Y 495.031,Z 628.449,A -85,B 0,C 180,E1 -6205.115,E2 -6205.115} C_VEL
LIN {X 0,Y 495.033,Z 631.837,A -85,B 0,C 180,E1 -6206.746,E2 -6206.746} C_VEL
LIN {X 0,Y 494.958,Z 633.838,A -85,B 0,C 180,E1 -6208.374,E2 -6208.374} C_VEL
LIN {X 0,Y 494.896,Z 634.5,A -85,B 0,C 180,E1 -6210.001,E2 -6210.001} C_VEL
LIN {X 0,Y 494.958,Z 633.834,A -85,B 0,C 180,E1 -6211.628,E2 -6211.628} C_VEL
LIN {X 0,Y 495.034,Z 631.83,A -85,B 0,C 180,E1 -6213.256,E2 -6213.256} C_VEL
LIN {X 0,Y 495.032,Z 628.441,A -85,B 0,C 180,E1 -6214.887,E2 -6214.887} C_VEL
LIN {X 0,Y 495.135,Z 624.515,A -85,B 0,C 180,E1 -6216.248,E2 -6216.248} C_VEL
LIN {X 0,Y 495.264,Z 618.859,A -85,B 0,C 180,E1 -6217.749,E2 -6217.749} C_VEL
LIN {X 0,Y 495.499,Z 612.028,A -85,B 0,C 180,E1 -6219.183,E2 -6219.183} C_VEL
LIN {X 0,Y 495.836,Z 603.549,A -85,B 0,C 180,E1 -6220.619,E2 -6220.619} C_VEL
LIN {X 0,Y 496.267,Z 593.764,A -85,B 0,C 180,E1 -6221.97,E2 -6221.97} C_VEL
LIN {X 0,Y 496.67,Z 583.976,A -85,B 0,C 180,E1 -6223.086,E2 -6223.086} C_VEL
LIN {X 0,Y 497.189,Z 573.121,A -85,B 0,C 180,E1 -6224.114,E2 -6224.114} C_VEL
LIN {X 0,Y 497.765,Z 561.232,A -85,B 0,C 180,E1 -6225.038,E2 -6225.038} C_VEL
LIN {X 0,Y 498.284,Z 548.082,A -85,B 0,C 180,E1 -6225.86,E2 -6225.86} C_VEL
LIN {X 0,Y 498.736,Z 535.172,A -85,B 0,C 180,E1 -6226.486,E2 -6226.486} C_VEL
LIN {X 0,Y 499.025,Z 521.359,A -85,B 0,C 180,E1 -6226.985,E2 -6226.985} C_VEL
LIN {X 0,Y 499.357,Z 507.077,A -85,B 0,C 180,E1 -6227.324,E2 -6227.324} C_VEL
LIN {X 0,Y 500.196,Z 387.815,A -85,B 0,C 180,E1 -6229.072,E2 -6229.072} C_VEL
LIN {X 0,Y 497.257,Z 372.428,A -85,B 0,C 180,E1 -6229.435,E2 -6229.435} C_VEL
LIN {X 0,Y 497.388,Z 367.082,A -85,B 0,C 180,E1 -6230.255,E2 -6230.255} C_VEL
LIN {X 0,Y 498.1,Z 350.081,A -85,B 0,C 180,E1 -6233.051,E2 -6233.051} C_VEL
LIN {X 0,Y 497.601,Z 346.072,A -85,B 0,C 180,E1 -6233.752,E2 -6233.752} C_VEL
LIN {X 0,Y 495.812,Z 337.437,A -85,B 0,C 180,E1 -6235.363,E2 -6235.363} C_VEL
LIN {X 0,Y 495.786,Z 337.347,A -85,B 0,C 180,E1 -6237.892,E2 -6237.892} C_VEL
LIN {X 0,Y 495.756,Z 337.356,A -85,B 0,C 180,E1 -6240.688,E2 -6240.688} C_VEL
LIN {X 0,Y 495.766,Z 337.354,A -85,B 0,C 180,E1 -6243.565,E2 -6243.565} C_VEL
LIN {X 0,Y 495.739,Z 337.359,A -85,B 0,C 180,E1 -6246.544,E2 -6246.544} C_VEL
LIN {X 0,Y 495.761,Z 337.356,A -85,B 0,C 180,E1 -6249.638,E2 -6249.638} C_VEL
LIN {X 0,Y 495.742,Z 337.355,A -85,B 0,C 180,E1 -6252.507,E2 -6252.507} C_VEL
LIN {X 0,Y 495.742,Z 337.355,A -85,B 0,C 180,E1 -6255.141,E2 -6255.141} C_VEL
LIN {X 0,Y 495.762,Z 337.357,A -85,B 0,C 180,E1 -6258.219,E2 -6258.219} C_VEL
LIN {X 0,Y 495.754,Z 337.357,A -85,B 0,C 180,E1 -6261.409,E2 -6261.409} C_VEL
LIN {X 0,Y 495.752,Z 337.356,A -85,B 0,C 180,E1 -6264.463,E2 -6264.463} C_VEL
LIN {X 0,Y 495.772,Z 337.357,A -85,B 0,C 180,E1 -6267.406,E2 -6267.406} C_VEL
LIN {X 0,Y 495.771,Z 337.357,A -85,B 0,C 180,E1 -6270.254,E2 -6270.254} C_VEL
LIN {X 0,Y 495.837,Z 337.504,A -85,B 0,C 180,E1 -6272.856,E2 -6272.856} C_VEL
LIN {X 0,Y 498.139,Z 349.255,A -85,B 0,C 180,E1 -6274.549,E2 -6274.549} C_VEL
LIN {X 0,Y 497.754,Z 370.738,A -85,B 0,C 180,E1 -6277.372,E2 -6277.372} C_VEL
LIN {X 0,Y 497.347,Z 390.291,A -85,B 0,C 180,E1 -6279.96,E2 -6279.96} C_VEL
LIN {X 0,Y 496.878,Z 412.655,A -85,B 0,C 180,E1 -6282.933,E2 -6282.933} C_VEL
LIN {X 0,Y 496.727,Z 421.002,A -85,B 0,C 180,E1 -6284.019,E2 -6284.019} C_VEL
LIN {X 0,Y 498.463,Z 433.517,A -85,B 0,C 180,E1 -6284.303,E2 -6284.303} C_VEL
LIN {X 0,Y 497.668,Z 532.034,A -85,B 0,C 180,E1 -6285.875,E2 -6285.875} C_VEL
LIN {X 0,Y 497.448,Z 543.963,A -85,B 0,C 180,E1 -6286.207,E2 -6286.207} C_VEL
LIN {X 0,Y 497.131,Z 556.496,A -85,B 0,C 180,E1 -6286.719,E2 -6286.719} C_VEL
LIN {X 0,Y 496.808,Z 569.111,A -85,B 0,C 180,E1 -6287.413,E2 -6287.413} C_VEL
LIN {X 0,Y 496.48,Z 580.86,A -85,B 0,C 180,E1 -6288.259,E2 -6288.259} C_VEL
LIN {X 0,Y 496.096,Z 591.129,A -85,B 0,C 180,E1 -6289.181,E2 -6289.181} C_VEL
LIN {X 0,Y 495.803,Z 600.416,A -85,B 0,C 180,E1 -6290.206,E2 -6290.206} C_VEL
LIN {X 0,Y 495.513,Z 609.349,A -85,B 0,C 180,E1 -6291.435,E2 -6291.435} C_VEL
LIN {X 0,Y 495.276,Z 616.549,A -85,B 0,C 180,E1 -6292.663,E2 -6292.663} C_VEL
LIN {X 0,Y 495.169,Z 622.792,A -85,B 0,C 180,E1 -6294.017,E2 -6294.017} C_VEL
LIN {X 0,Y 495.021,Z 628.002,A -85,B 0,C 180,E1 -6295.522,E2 -6295.522} C_VEL
LIN {X 0,Y 495.043,Z 631.034,A -85,B 0,C 180,E1 -6296.745,E2 -6296.745} C_VEL
LIN {X 0,Y 494.975,Z 632.517,A -85,B 0,C 180,E1 -6297.559,E2 -6297.559} C_VEL
LIN {X 0,Y 494.962,Z 633.546,A -85,B 0,C 180,E1 -6298.373,E2 -6298.373} C_VEL
LIN {X 0,Y 494.899,Z 634.43,A -85,B 0,C 180,E1 -6300,E2 -6300} C_VEL
LIN {X 0,Y 494.911,Z 634.238,A -85,B 0,C 180,E1 -6300.814,E2 -6300.814} C_VEL
LIN {X 0,Y 494.962,Z 633.638,A -85,B 0,C 180,E1 -6301.627,E2 -6301.627} C_VEL
LIN {X 0,Y 494.975,Z 632.648,A -85,B 0,C 180,E1 -6302.441,E2 -6302.441} C_VEL
LIN {X 0,Y 495.043,Z 631.242,A -85,B 0,C 180,E1 -6303.255,E2 -6303.255} C_VEL
LIN {X 0,Y 495.021,Z 628.294,A -85,B 0,C 180,E1 -6304.479,E2 -6304.479} C_VEL
LIN {X 0,Y 495.159,Z 623.195,A -85,B 0,C 180,E1 -6305.981,E2 -6305.981} C_VEL
LIN {X 0,Y 495.275,Z 617.102,A -85,B 0,C 180,E1 -6307.337,E2 -6307.337} C_VEL
LIN {X 0,Y 495.503,Z 610.066,A -85,B 0,C 180,E1 -6308.565,E2 -6308.565} C_VEL
LIN {X 0,Y 495.747,Z 601.301,A -85,B 0,C 180,E1 -6309.795,E2 -6309.795} C_VEL
LIN {X 0,Y 496.073,Z 592.308,A -85,B 0,C 180,E1 -6310.82,E2 -6310.82} C_VEL
LIN {X 0,Y 496.485,Z 582.348,A -85,B 0,C 180,E1 -6311.741,E2 -6311.741} C_VEL
LIN {X 0,Y 496.789,Z 570.939,A -85,B 0,C 180,E1 -6312.593,E2 -6312.593} C_VEL
LIN {X 0,Y 497.146,Z 559.154,A -85,B 0,C 180,E1 -6313.281,E2 -6313.281} C_VEL
LIN {X 0,Y 497.493,Z 546.136,A -85,B 0,C 180,E1 -6313.844,E2 -6313.844} C_VEL
LIN {X 0,Y 497.766,Z 533.381,A -85,B 0,C 180,E1 -6314.227,E2 -6314.227} C_VEL
LIN {X 0,Y 497.924,Z 513.645,A -85,B 0,C 180,E1 -6314.561,E2 -6314.561} C_VEL
LIN {X 0,Y 498.372,Z 432.193,A -85,B 0,C 180,E1 -6315.828,E2 -6315.828} C_VEL
LIN {X 0,Y 496.724,Z 420.949,A -85,B 0,C 180,E1 -6316.085,E2 -6316.085} C_VEL
LIN {X 0,Y 497.287,Z 398.106,A -85,B 0,C 180,E1 -6319.183,E2 -6319.183} C_VEL
LIN {X 0,Y 497.886,Z 376.155,A -85,B 0,C 180,E1 -6322.185,E2 -6322.185} C_VEL
LIN {X 0,Y 498.491,Z 355.511,A -85,B 0,C 180,E1 -6325.022,E2 -6325.022} C_VEL
LIN {X 0,Y 498.527,Z 350.863,A -85,B 0,C 180,E1 -6325.667,E2 -6325.667} C_VEL
LIN {X 0,Y 496.192,Z 339.132,A -85,B 0,C 180,E1 -6327.408,E2 -6327.408} C_VEL
LIN {X 0,Y 495.844,Z 337.445,A -85,B 0,C 180,E1 -6327.715,E2 -6327.715} C_VEL
LIN {X 0,Y 495.757,Z 337.36,A -85,B 0,C 180,E1 -6330.687,E2 -6330.687} C_VEL
LIN {X 0,Y 495.764,Z 337.353,A -85,B 0,C 180,E1 -6333.564,E2 -6333.564} C_VEL
LIN {X 0,Y 495.733,Z 337.362,A -85,B 0,C 180,E1 -6336.544,E2 -6336.544} C_VEL
LIN {X 0,Y 495.761,Z 337.353,A -85,B 0,C 180,E1 -6339.638,E2 -6339.638} C_VEL
LIN {X 0,Y 495.76,Z 337.352,A -85,B 0,C 180,E1 -6341.294,E2 -6341.294} C_VEL
LIN {X 0,Y 495.085,Z 337.442,A -85,B 0,C 180,E1 -6341.972,E2 -6341.972} C_VEL
LIN {X 0,Y 492.231,Z 337.79,A -85,B 0,C 180,E1 -6343.073,E2 -6343.073} C_VEL
LIN {X 0,Y 489.823,Z 338.091,A -85,B 0,C 180,E1 -6343.961,E2 -6343.961} C_VEL
LIN {X 0,Y 488.789,Z 338.213,A -85,B 0,C 180,E1 -6344.646,E2 -6344.646} C_VEL
LIN {X 0,Y 488.705,Z 338.222,A -85,B 0,C 180,E1 -6344.878,E2 -6344.878} C_VEL
LIN {X 0,Y 488.697,Z 338.233,A -85,B 0,C 180,E1 -6347.474,E2 -6347.474} C_VEL
LIN {X 0,Y 488.738,Z 338.228,A -85,B 0,C 180,E1 -6349.676,E2 -6349.676} C_VEL
LIN {X 0,Y 488.687,Z 338.234,A -85,B 0,C 180,E1 -6352.841,E2 -6352.841} C_VEL
LIN {X 0,Y 488.74,Z 338.234,A -85,B 0,C 180,E1 -6355.887,E2 -6355.887} C_VEL
LIN {X 0,Y 488.697,Z 338.234,A -85,B 0,C 180,E1 -6358.82,E2 -6358.82} C_VEL
LIN {X 0,Y 488.75,Z 338.215,A -85,B 0,C 180,E1 -6361.671,E2 -6361.671} C_VEL
LIN {X 0,Y 488.818,Z 338.312,A -85,B 0,C 180,E1 -6364.447,E2 -6364.447} C_VEL
LIN {X 0,Y 491.044,Z 349.477,A -85,B 0,C 180,E1 -6366.54,E2 -6366.54} C_VEL
LIN {X 0,Y 491.047,Z 355.044,A -85,B 0,C 180,E1 -6367.489,E2 -6367.489} C_VEL
LIN {X 0,Y 490.327,Z 372.206,A -85,B 0,C 180,E1 -6370.309,E2 -6370.309} C_VEL
LIN {X 0,Y 492.778,Z 384.982,A -85,B 0,C 180,E1 -6370.633,E2 -6370.633} C_VEL
LIN {X 0,Y 493.542,Z 390.368,A -85,B 0,C 180,E1 -6370.745,E2 -6370.745} C_VEL
LIN {X 0,Y 492.576,Z 509.023,A -85,B 0,C 180,E1 -6372.51,E2 -6372.51} C_VEL
LIN {X 0,Y 492.229,Z 523.331,A -85,B 0,C 180,E1 -6372.882,E2 -6372.882} C_VEL
LIN {X 0,Y 491.864,Z 536.731,A -85,B 0,C 180,E1 -6373.394,E2 -6373.394} C_VEL
LIN {X 0,Y 491.4,Z 549.11,A -85,B 0,C 180,E1 -6374.018,E2 -6374.018} C_VEL
LIN {X 0,Y 490.835,Z 562.054,A -85,B 0,C 180,E1 -6374.851,E2 -6374.851} C_VEL
LIN {X 0,Y 490.261,Z 573.796,A -85,B 0,C 180,E1 -6375.788,E2 -6375.788} C_VEL
LIN {X 0,Y 489.645,Z 585.51,A -85,B 0,C 180,E1 -6376.934,E2 -6376.934} C_VEL
LIN {X 0,Y 489.255,Z 594.955,A -85,B 0,C 180,E1 -6378.055,E2 -6378.055} C_VEL
LIN {X 0,Y 488.749,Z 604.612,A -85,B 0,C 180,E1 -6379.435,E2 -6379.435} C_VEL
LIN {X 0,Y 488.452,Z 612.892,A -85,B 0,C 180,E1 -6380.892,E2 -6380.892} C_VEL
LIN {X 0,Y 488.205,Z 618.663,A -85,B 0,C 180,E1 -6382.139,E2 -6382.139} C_VEL
LIN {X 0,Y 488.039,Z 624.765,A -85,B 0,C 180,E1 -6383.781,E2 -6383.781} C_VEL
LIN {X 0,Y 487.963,Z 628.325,A -85,B 0,C 180,E1 -6385.042,E2 -6385.042} C_VEL
